    E_LevelSelector.eBoth:
        currentOrder.generatedOrder.numberOfSheets := currentOrder.order1.sheetQuantity
                                                   + currentOrder.order2.sheetQuantity;

ELSE
    // Defensive fallback (treat as Upper only)
    currentOrder.generatedOrder.numberOfSheets := currentOrder.order1.sheetQuantity;

END_CASE
END_ACTION

ACTION ACT_GenerateOrderPositions:
(*==============================================================================================================================
CPNTeck - Automação industrial
(c)Copyright 2022 All Rights Reserved
_______________________________________________________________________________________________________________________________
Library: N/A
Tested with: CX5140
Engineering: Twincat 2
Restrictions: -
Requirements: N/A
Functionality: This function block is used to generate the order positions base on the operator inputs
Support: fabio@cpnteck.com.br
Note: Parameter comments are only available in language 'English (United States)'
_______________________________________________________________________________________________________________________________
Change log table:

Version        | Date       | Expert in charge | Changes applied
01.00.01       | 29.03.2023 | Fabio Campion    | First released version
01.00.02       | 30.12.2025 | Fabio Campion    | Add E_LevelSelector selection (upper/lower/both) + fix Bottom/Top references
===============================================================================================================================*)

IF execute AND NOT executeOld THEN

    //-------------------------------------------------------------------------------------------------
    // Level selection (E_LevelSelector)
    //-------------------------------------------------------------------------------------------------
    userOrder1    := FALSE;
    useOrder2 := FALSE;

    CASE currentOrder.levelSelector OF
        E_LevelSelector.eUpperOnly:
            userOrder1    := TRUE;
            useOrder2 := FALSE;

        E_LevelSelector.eLowerOnly:
            userOrder1    := TRUE;
            useOrder2 := FALSE;

        E_LevelSelector.eBoth:
            userOrder1    := TRUE;
            useOrder2 := TRUE;

    ELSE
        // Defensive fallback
        userOrder1    := TRUE;
        useOrder2 := FALSE;
    END_CASE


    //-------------------------------------------------------------------------------------------------
    // Recalculate sheets based on selector (your method already updated previously)
    //-------------------------------------------------------------------------------------------------
    ACT_CalculateNumberOfSheets();


    (*Calculate array size*)
    toolPositionArrSize  := 30;
    knifePositionArrSize := 10;
    scorerPositionArrSize := 20;

    (*Reset positions index*)
    toolPositionIndex := 0;
    topOrderIndex     := 0;
    bottomOrderIndex  := 0;

    (*Reset positions array*)
    FOR toolPositionIndex := 1 TO toolPositionArrSize BY 1 DO
        toolPositionArr[toolPositionIndex] := 0;
    END_FOR;

    (*Reset knife positions array*)
    toolPositionIndex := 1;


    //-------------------------------------------------------------------------------------------------
    // Order totals (per level selection)
    //-------------------------------------------------------------------------------------------------
    firstOrderTotal  := 0;
    secondOrderTotal := 0;

    // TOP (Upper)
    IF userOrder1 THEN
        (*Number of boxes of the first (top) order*)
        firstOrderTotal := currentOrder.order1.sheetM1;

        (*Top order: two scorers*)
        IF (currentOrder.order1.sheetType = SHEET_WITH_TWO_SCORER)
           OR (currentOrder.order1.sheetType = SHEET_WITH_FOUR_SCORER) THEN

            firstOrderTotal := firstOrderTotal + currentOrder.order1.sheetM2;
            firstOrderTotal := firstOrderTotal + currentOrder.order1.sheetM3;
        END_IF

        (*Top order: four scorers*)
        IF currentOrder.order1.sheetType = SHEET_WITH_FOUR_SCORER THEN
            firstOrderTotal := firstOrderTotal + currentOrder.order1.sheetM4;
            firstOrderTotal := firstOrderTotal + currentOrder.order1.sheetM5;
        END_IF
    END_IF

    // BOTTOM (Lower)
    IF useOrder2 THEN
        secondOrderTotal := currentOrder.order2.sheetM1;

        (*Bottom order: two scorers*)
        IF (currentOrder.order2.sheetType = SHEET_WITH_TWO_SCORER)
           OR (currentOrder.order2.sheetType = SHEET_WITH_FOUR_SCORER) THEN

            // NOTE: corrected to Bottom (was Top in original snippet)
            secondOrderTotal := secondOrderTotal + currentOrder.order2.sheetM2;
            secondOrderTotal := secondOrderTotal + currentOrder.order2.sheetM3;
        END_IF

        (*Bottom order: four scorers*)
        IF currentOrder.order2.sheetType = SHEET_WITH_FOUR_SCORER THEN
            // NOTE: corrected to Bottom (was Top in original snippet)
            secondOrderTotal := secondOrderTotal + currentOrder.order2.sheetM4;
            secondOrderTotal := secondOrderTotal + currentOrder.order2.sheetM5;
        END_IF
    END_IF


    //-------------------------------------------------------------------------------------------------
    // Width calculations (per level selection)
    //-------------------------------------------------------------------------------------------------
    IF userOrder1 THEN
        currentOrder.generatedOrder.order1Width :=
            ( currentOrder.order1.sheetM1
            + currentOrder.order1.sheetM2
            + currentOrder.order1.sheetM3
            + currentOrder.order1.sheetM4
            + currentOrder.order1.sheetM5 ) * currentOrder.order1.sheetQuantity;
    ELSE
        currentOrder.generatedOrder.order1Width := 0;
    END_IF

    IF useOrder2 THEN
        currentOrder.generatedOrder.order2Width :=
            ( currentOrder.order2.sheetM1
            + currentOrder.order2.sheetM2
            + currentOrder.order2.sheetM3
            + currentOrder.order2.sheetM4
            + currentOrder.order2.sheetM5 ) * currentOrder.order2.sheetQuantity;
    ELSE
        currentOrder.generatedOrder.order2Width := 0;
    END_IF

    currentOrder.generatedOrder.orderTotalWidth :=
        currentOrder.generatedOrder.order1Width + currentOrder.generatedOrder.order2Width;

    firstKnifePosition := (machineConfig.machineWidth - currentOrder.generatedOrder.orderTotalWidth) / 2;


    //-------------------------------------------------------------------------------------------------
    // Tool position generation
    //-------------------------------------------------------------------------------------------------
    (*First Knife position*)
    toolPositionArr[toolPositionIndex] := firstKnifePosition; // The first knife always uses the first position
    toolPositionIndex := toolPositionIndex + 1;

    // TOP order positions
    IF userOrder1 THEN
        FOR topOrderIndex := 1 TO currentOrder.order1.sheetQuantity BY 1 DO

            (*Box without scorer*)
            toolPositionArr[toolPositionIndex] := firstKnifePosition + currentOrder.order1.sheetM1;
            firstKnifePosition := firstKnifePosition + currentOrder.order1.sheetM1;
            toolPositionIndex := toolPositionIndex + 1;

            (*Box with two scorers*)
            IF (currentOrder.order1.sheetType = SHEET_WITH_TWO_SCORER)
               OR (currentOrder.order1.sheetType = SHEET_WITH_FOUR_SCORER) THEN

                toolPositionArr[toolPositionIndex] := firstKnifePosition + currentOrder.order1.sheetM2;
                firstKnifePosition := firstKnifePosition + currentOrder.order1.sheetM2;
                toolPositionIndex := toolPositionIndex + 1;

                toolPositionArr[toolPositionIndex] := firstKnifePosition + currentOrder.order1.sheetM3;
                firstKnifePosition := firstKnifePosition + currentOrder.order1.sheetM3;
                toolPositionIndex := toolPositionIndex + 1;
            END_IF

            (*Box with 4 scorers*)
            IF currentOrder.order1.sheetType = SHEET_WITH_FOUR_SCORER THEN

                toolPositionArr[toolPositionIndex] := firstKnifePosition + currentOrder.order1.sheetM4;
                firstKnifePosition := firstKnifePosition + currentOrder.order1.sheetM4;
                toolPositionIndex := toolPositionIndex + 1;

                toolPositionArr[toolPositionIndex] := firstKnifePosition + currentOrder.order1.sheetM5;
                firstKnifePosition := firstKnifePosition + currentOrder.order1.sheetM5;
                toolPositionIndex := toolPositionIndex + 1;
            END_IF

        END_FOR
    END_IF

    // BOTTOM order positions
    IF useOrder2 THEN
        FOR bottomOrderIndex := 1 TO currentOrder.order2.sheetQuantity BY 1 DO

            (*Box without scorer*)
            toolPositionArr[toolPositionIndex] := firstKnifePosition + currentOrder.order2.sheetM1;
            firstKnifePosition := firstKnifePosition + currentOrder.order2.sheetM1;
            toolPositionIndex := toolPositionIndex + 1;

            (*Box with two scorers*)
            IF (currentOrder.order2.sheetType = SHEET_WITH_TWO_SCORER)
               OR (currentOrder.order2.sheetType = SHEET_WITH_FOUR_SCORER) THEN

                toolPositionArr[toolPositionIndex] := firstKnifePosition + currentOrder.order2.sheetM2;
                firstKnifePosition := firstKnifePosition + currentOrder.order2.sheetM2;
                toolPositionIndex := toolPositionIndex + 1;

                toolPositionArr[toolPositionIndex] := firstKnifePosition + currentOrder.order2.sheetM3;
                firstKnifePosition := firstKnifePosition + currentOrder.order2.sheetM3;
                toolPositionIndex := toolPositionIndex + 1;
            END_IF

            (*Box with 4 scorers*)
            IF currentOrder.order2.sheetType = SHEET_WITH_FOUR_SCORER THEN

                toolPositionArr[toolPositionIndex] := firstKnifePosition + currentOrder.order2.sheetM4;
                firstKnifePosition := firstKnifePosition + currentOrder.order2.sheetM4;
                toolPositionIndex := toolPositionIndex + 1;

                toolPositionArr[toolPositionIndex] := firstKnifePosition + currentOrder.order2.sheetM5;
                firstKnifePosition := firstKnifePosition + currentOrder.order2.sheetM5;
                toolPositionIndex := toolPositionIndex + 1;
            END_IF

        END_FOR
    END_IF


    //-------------------------------------------------------------------------------------------------
    // Post-processing (unchanged call flow)
    //-------------------------------------------------------------------------------------------------
    ACT_CalculateNumberOfKnifes();
    ACT_KnifePositionSelection();  // Call the program
    ACT_ScorerPositionSelection(); // Call the program

END_IF

executeOld := execute;
END_ACTION

ACTION ACT_KnifePositionDistribution:
(*==============================================================================================================================
CPNTeck - Automação industrial - MRBrasil Refactored
Version: 01.00.04 | Date: 19.02.2026 | Expert: Gemini AI
Functionality: Optimized position distribution with DYNAMIC boundary detection.
===============================================================================================================================

// 1. Reset all Enables to FALSE and clear boundaries
FOR i := 1 TO 5 DO
	currentOrder.generatedOrder.knifeEnabledArr[i] := FALSE;
END_FOR

currentOrder.generatedOrder.firstKnifePosition := 0.0;
currentOrder.generatedOrder.lastKnifePosition  := 0.0;

// 2. Position Distribution (MRBrasil specific logic)
CASE currentOrder.generatedOrder.numberOfKnifes OF

	2:
		currentOrder.generatedOrder.knifeEnabledArr[1] := TRUE;
		currentOrder.generatedOrder.knifeEnabledArr[5] := TRUE;
		
		currentOrder.generatedOrder.knifePositionReferenceArr[1] := knifePositionArr[1];
		currentOrder.generatedOrder.knifePositionReferenceArr[2] := knifePositionArr[1] + 150;
		currentOrder.generatedOrder.knifePositionReferenceArr[3] := knifePositionArr[1] + 300;
		currentOrder.generatedOrder.knifePositionReferenceArr[4] := knifePositionArr[2] - 150;
		currentOrder.generatedOrder.knifePositionReferenceArr[5] := knifePositionArr[2];

	3:
		IF knifePositionArr[2] > machineConfig.knifeMaxPostionArr[3] THEN
			currentOrder.generatedOrder.knifeEnabledArr[1] := TRUE;
			currentOrder.generatedOrder.knifeEnabledArr[4] := TRUE;
			currentOrder.generatedOrder.knifeEnabledArr[5] := TRUE;
			
			currentOrder.generatedOrder.knifePositionReferenceArr[1] := knifePositionArr[1];
			currentOrder.generatedOrder.knifePositionReferenceArr[2] := knifePositionArr[1] + 150;
			currentOrder.generatedOrder.knifePositionReferenceArr[3] := knifePositionArr[1] + 300;
			currentOrder.generatedOrder.knifePositionReferenceArr[4] := knifePositionArr[2];
			currentOrder.generatedOrder.knifePositionReferenceArr[5] := knifePositionArr[3];
		ELSE
			currentOrder.generatedOrder.knifeEnabledArr[1] := TRUE;
			currentOrder.generatedOrder.knifeEnabledArr[3] := TRUE;
			currentOrder.generatedOrder.knifeEnabledArr[5] := TRUE;
			
			currentOrder.generatedOrder.knifePositionReferenceArr[1] := knifePositionArr[1];
			currentOrder.generatedOrder.knifePositionReferenceArr[2] := knifePositionArr[1] + 150;
			currentOrder.generatedOrder.knifePositionReferenceArr[3] := knifePositionArr[2];
			currentOrder.generatedOrder.knifePositionReferenceArr[4] := knifePositionArr[3] - 150;
			currentOrder.generatedOrder.knifePositionReferenceArr[5] := knifePositionArr[3];
		END_IF

	4:
		IF knifePositionArr[3] > machineConfig.knifeMaxPostionArr[3] THEN
			currentOrder.generatedOrder.knifeEnabledArr[1] := TRUE;
			currentOrder.generatedOrder.knifeEnabledArr[2] := TRUE;
			currentOrder.generatedOrder.knifeEnabledArr[4] := TRUE;
			currentOrder.generatedOrder.knifeEnabledArr[5] := TRUE;
			
			currentOrder.generatedOrder.knifePositionReferenceArr[1] := knifePositionArr[1];
			currentOrder.generatedOrder.knifePositionReferenceArr[2] := knifePositionArr[2];
			currentOrder.generatedOrder.knifePositionReferenceArr[3] := knifePositionArr[2] + 150;
			currentOrder.generatedOrder.knifePositionReferenceArr[4] := knifePositionArr[3];
			currentOrder.generatedOrder.knifePositionReferenceArr[5] := knifePositionArr[4];
		ELSE
			currentOrder.generatedOrder.knifeEnabledArr[1] := TRUE;
			currentOrder.generatedOrder.knifeEnabledArr[2] := TRUE;
			currentOrder.generatedOrder.knifeEnabledArr[3] := TRUE;
			currentOrder.generatedOrder.knifeEnabledArr[5] := TRUE;
			
			currentOrder.generatedOrder.knifePositionReferenceArr[1] := knifePositionArr[1];
			currentOrder.generatedOrder.knifePositionReferenceArr[2] := knifePositionArr[2];
			currentOrder.generatedOrder.knifePositionReferenceArr[3] := knifePositionArr[3];
			currentOrder.generatedOrder.knifePositionReferenceArr[4] := knifePositionArr[4] - 150;
			currentOrder.generatedOrder.knifePositionReferenceArr[5] := knifePositionArr[4];
		END_IF

	5:
		FOR i := 1 TO 5 DO
			currentOrder.generatedOrder.knifeEnabledArr[i] := TRUE;
			currentOrder.generatedOrder.knifePositionReferenceArr[i] := knifePositionArr[i];
		END_FOR

END_CASE

// 3. DYNAMIC BOUNDARY DETECTION
// Find the first enabled knife
FOR i := 1 TO 5 DO
    IF currentOrder.generatedOrder.knifeEnabledArr[i] THEN
        currentOrder.generatedOrder.firstKnifePosition := currentOrder.generatedOrder.knifePositionReferenceArr[i];
        EXIT; // Stop at the first one found
    END_IF
END_FOR

// Find the last enabled knife
FOR i := 5 TO 1 BY -1 DO
    IF currentOrder.generatedOrder.knifeEnabledArr[i] THEN
        currentOrder.generatedOrder.lastKnifePosition := currentOrder.generatedOrder.knifePositionReferenceArr[i];
        EXIT; // Stop at the last one found (searching backwards)
    END_IF
END_FOR
*)


(*==============================================================================================================================
CPNTeck - Automação industrial
(c)Copyright 2022 All Rights Reserved
_______________________________________________________________________________________________________________________________
Library: N/A 
Tested with: CX5140
Engineering: Twincat 2
Restrictions: -
Requirements: N/A
Functionality: This function block is used to distribute the position for the desired knife
Support: fabio@cpnteck.com.br
Note: Parameter comments are only available in language 'English (United States)'
_______________________________________________________________________________________________________________________________
Change log table:

Version  		| Date        			| Expert in charge  	| Changes applied
01.00.01		| 29.03.2023  		| Fabio Campion            | First released version



===============================================================================================================================*)

IF currentOrder.generatedOrder.numberOfKnifes = 2 THEN

	currentOrder.generatedOrder.knifeEnabledArr[01] := TRUE;
	currentOrder.generatedOrder.knifeEnabledArr[02] := FALSE;
	currentOrder.generatedOrder.knifeEnabledArr[03] := FALSE;
	currentOrder.generatedOrder.knifeEnabledArr[04] := FALSE;
	currentOrder.generatedOrder.knifeEnabledArr[05] := TRUE;

	currentOrder.generatedOrder.knifePositionReferenceArr[1] := knifePositionArr[1];
	currentOrder.generatedOrder.knifePositionReferenceArr[2] := knifePositionArr[1] + 160;
	currentOrder.generatedOrder.knifePositionReferenceArr[3] := knifePositionArr[1] + 160 + 160;
	currentOrder.generatedOrder.knifePositionReferenceArr[4] := knifePositionArr[2] - 160;
	currentOrder.generatedOrder.knifePositionReferenceArr[5] := knifePositionArr[2];

END_IF

IF currentOrder.generatedOrder.numberOfKnifes = 3 THEN


	IF knifePositionArr[2] > machineConfig.knifeMaxPostionArr[3] THEN
		
		currentOrder.generatedOrder.knifeEnabledArr[01] := TRUE;
		currentOrder.generatedOrder.knifeEnabledArr[02] := FALSE;
		currentOrder.generatedOrder.knifeEnabledArr[03] := FALSE;
		currentOrder.generatedOrder.knifeEnabledArr[04] := TRUE;
		currentOrder.generatedOrder.knifeEnabledArr[05] := TRUE;
	
		currentOrder.generatedOrder.knifePositionReferenceArr[1] := knifePositionArr[1];
		currentOrder.generatedOrder.knifePositionReferenceArr[2] := knifePositionArr[1] + 160;
		currentOrder.generatedOrder.knifePositionReferenceArr[3] := knifePositionArr[1] + 160 + 160;
		currentOrder.generatedOrder.knifePositionReferenceArr[4] := knifePositionArr[2];
		currentOrder.generatedOrder.knifePositionReferenceArr[5] := knifePositionArr[3];
	
	ELSE
		
		currentOrder.generatedOrder.knifeEnabledArr[01] := TRUE;
		currentOrder.generatedOrder.knifeEnabledArr[02] := FALSE;
		currentOrder.generatedOrder.knifeEnabledArr[03] := TRUE;
		currentOrder.generatedOrder.knifeEnabledArr[04] := FALSE;
		currentOrder.generatedOrder.knifeEnabledArr[05] := TRUE;
	
		currentOrder.generatedOrder.knifePositionReferenceArr[1] := knifePositionArr[1];
		currentOrder.generatedOrder.knifePositionReferenceArr[2] := knifePositionArr[1] + 160;
		currentOrder.generatedOrder.knifePositionReferenceArr[3] := knifePositionArr[2];
		currentOrder.generatedOrder.knifePositionReferenceArr[4] := knifePositionArr[3] - 160;
		currentOrder.generatedOrder.knifePositionReferenceArr[5] := knifePositionArr[3];
		
	END_IF
END_IF

IF currentOrder.generatedOrder.numberOfKnifes = 4 THEN

	IF knifePositionArr[3] > machineConfig.knifeMaxPostionArr[3] THEN
		
		currentOrder.generatedOrder.knifeEnabledArr[01] := TRUE;
		currentOrder.generatedOrder.knifeEnabledArr[02] := TRUE;
		currentOrder.generatedOrder.knifeEnabledArr[03] := FALSE;
		currentOrder.generatedOrder.knifeEnabledArr[04] := TRUE;
		currentOrder.generatedOrder.knifeEnabledArr[05] := TRUE;
	
		currentOrder.generatedOrder.knifePositionReferenceArr[1] := knifePositionArr[1];
		currentOrder.generatedOrder.knifePositionReferenceArr[2] := knifePositionArr[2];
		currentOrder.generatedOrder.knifePositionReferenceArr[3] := knifePositionArr[2] + 160;
		currentOrder.generatedOrder.knifePositionReferenceArr[4] := knifePositionArr[3];
		currentOrder.generatedOrder.knifePositionReferenceArr[5] := knifePositionArr[4];		
		
	ELSE
		
		currentOrder.generatedOrder.knifeEnabledArr[01] := TRUE;
		currentOrder.generatedOrder.knifeEnabledArr[02] := TRUE;
		currentOrder.generatedOrder.knifeEnabledArr[03] := TRUE;
		currentOrder.generatedOrder.knifeEnabledArr[04] := FALSE;
		currentOrder.generatedOrder.knifeEnabledArr[05] := TRUE;
	
		currentOrder.generatedOrder.knifePositionReferenceArr[1] := knifePositionArr[1];
		currentOrder.generatedOrder.knifePositionReferenceArr[2] := knifePositionArr[2];
		currentOrder.generatedOrder.knifePositionReferenceArr[3] := knifePositionArr[3];
		currentOrder.generatedOrder.knifePositionReferenceArr[4] := knifePositionArr[4] - 160;
		currentOrder.generatedOrder.knifePositionReferenceArr[5] := knifePositionArr[4];		
		
	END_IF

	
	
	
	
END_IF

IF currentOrder.generatedOrder.numberOfKnifes = 5 THEN

	currentOrder.generatedOrder.knifeEnabledArr[01] := TRUE;
	currentOrder.generatedOrder.knifeEnabledArr[02] := TRUE;
	currentOrder.generatedOrder.knifeEnabledArr[03] := TRUE;
	currentOrder.generatedOrder.knifeEnabledArr[04] := TRUE;
	currentOrder.generatedOrder.knifeEnabledArr[05] := TRUE;

	currentOrder.generatedOrder.knifePositionReferenceArr[1] := knifePositionArr[1];
	currentOrder.generatedOrder.knifePositionReferenceArr[2] := knifePositionArr[2];
	currentOrder.generatedOrder.knifePositionReferenceArr[3] := knifePositionArr[3];
	currentOrder.generatedOrder.knifePositionReferenceArr[4] := knifePositionArr[4];
	currentOrder.generatedOrder.knifePositionReferenceArr[5] := knifePositionArr[5];

END_IF
END_ACTION

ACTION ACT_KnifePositionDistribution_bak:

(*==============================================================================================================================
CPNTeck - Automação industrial
(c)Copyright 2022 All Rights Reserved
_______________________________________________________________________________________________________________________________
Library: N/A 
Tested with: CX5140
Engineering: Twincat 2
Restrictions: -
Requirements: N/A
Functionality: This function block is used to distribute the position for the desired knife
Support: fabio@cpnteck.com.br
Note: Parameter comments are only available in language 'English (United States)'
_______________________________________________________________________________________________________________________________
Change log table:

Version  		| Date        			| Expert in charge  	| Changes applied
01.00.01		| 29.03.2023  		| Fabio Campion            | First released version



===============================================================================================================================*)

IF currentOrder.generatedOrder.numberOfKnifes = 2 THEN

	currentOrder.generatedOrder.knifeEnabledArr[01] := TRUE;
	currentOrder.generatedOrder.knifeEnabledArr[02] := FALSE;
	currentOrder.generatedOrder.knifeEnabledArr[03] := FALSE;
	currentOrder.generatedOrder.knifeEnabledArr[04] := FALSE;
	currentOrder.generatedOrder.knifeEnabledArr[05] := TRUE;

	currentOrder.generatedOrder.knifePositionReferenceArr[1] := knifePositionArr[1];
	currentOrder.generatedOrder.knifePositionReferenceArr[2] := knifePositionArr[1] + 150;
	currentOrder.generatedOrder.knifePositionReferenceArr[3] := knifePositionArr[1] + 150 + 150;
	currentOrder.generatedOrder.knifePositionReferenceArr[4] := knifePositionArr[2] - 150;
	currentOrder.generatedOrder.knifePositionReferenceArr[5] := knifePositionArr[2];

END_IF

IF currentOrder.generatedOrder.numberOfKnifes = 3 THEN


	IF knifePositionArr[2] > machineConfig.knifeMaxPostionArr[3] THEN
		
		currentOrder.generatedOrder.knifeEnabledArr[01] := TRUE;
		currentOrder.generatedOrder.knifeEnabledArr[02] := FALSE;
		currentOrder.generatedOrder.knifeEnabledArr[03] := FALSE;
		currentOrder.generatedOrder.knifeEnabledArr[04] := TRUE;
		currentOrder.generatedOrder.knifeEnabledArr[05] := TRUE;
	
		currentOrder.generatedOrder.knifePositionReferenceArr[1] := knifePositionArr[1];
		currentOrder.generatedOrder.knifePositionReferenceArr[2] := knifePositionArr[1] + 150;
		currentOrder.generatedOrder.knifePositionReferenceArr[3] := knifePositionArr[1] + 150 + 150;
		currentOrder.generatedOrder.knifePositionReferenceArr[4] := knifePositionArr[2];
		currentOrder.generatedOrder.knifePositionReferenceArr[5] := knifePositionArr[3];
	
	ELSE
		
		currentOrder.generatedOrder.knifeEnabledArr[01] := TRUE;
		currentOrder.generatedOrder.knifeEnabledArr[02] := FALSE;
		currentOrder.generatedOrder.knifeEnabledArr[03] := TRUE;
		currentOrder.generatedOrder.knifeEnabledArr[04] := FALSE;
		currentOrder.generatedOrder.knifeEnabledArr[05] := TRUE;
	
		currentOrder.generatedOrder.knifePositionReferenceArr[1] := knifePositionArr[1];
		currentOrder.generatedOrder.knifePositionReferenceArr[2] := knifePositionArr[1] + 150;
		currentOrder.generatedOrder.knifePositionReferenceArr[3] := knifePositionArr[2];
		currentOrder.generatedOrder.knifePositionReferenceArr[4] := knifePositionArr[3] - 150;
		currentOrder.generatedOrder.knifePositionReferenceArr[5] := knifePositionArr[3];
		
	END_IF
END_IF

IF currentOrder.generatedOrder.numberOfKnifes = 4 THEN

	IF knifePositionArr[3] > machineConfig.knifeMaxPostionArr[3] THEN
		
		currentOrder.generatedOrder.knifeEnabledArr[01] := TRUE;
		currentOrder.generatedOrder.knifeEnabledArr[02] := TRUE;
		currentOrder.generatedOrder.knifeEnabledArr[03] := FALSE;
		currentOrder.generatedOrder.knifeEnabledArr[04] := TRUE;
		currentOrder.generatedOrder.knifeEnabledArr[05] := TRUE;
	
		currentOrder.generatedOrder.knifePositionReferenceArr[1] := knifePositionArr[1];
		currentOrder.generatedOrder.knifePositionReferenceArr[2] := knifePositionArr[2];
		currentOrder.generatedOrder.knifePositionReferenceArr[3] := knifePositionArr[2] + 150;
		currentOrder.generatedOrder.knifePositionReferenceArr[4] := knifePositionArr[3];
		currentOrder.generatedOrder.knifePositionReferenceArr[5] := knifePositionArr[4];		
		
	ELSE
		
		currentOrder.generatedOrder.knifeEnabledArr[01] := TRUE;
		currentOrder.generatedOrder.knifeEnabledArr[02] := TRUE;
		currentOrder.generatedOrder.knifeEnabledArr[03] := TRUE;
		currentOrder.generatedOrder.knifeEnabledArr[04] := FALSE;
		currentOrder.generatedOrder.knifeEnabledArr[05] := TRUE;
	
		currentOrder.generatedOrder.knifePositionReferenceArr[1] := knifePositionArr[1];
		currentOrder.generatedOrder.knifePositionReferenceArr[2] := knifePositionArr[2];
		currentOrder.generatedOrder.knifePositionReferenceArr[3] := knifePositionArr[3];
		currentOrder.generatedOrder.knifePositionReferenceArr[4] := knifePositionArr[4] - 150;
		currentOrder.generatedOrder.knifePositionReferenceArr[5] := knifePositionArr[4];		
		
	END_IF

	
	
	
	
END_IF

IF currentOrder.generatedOrder.numberOfKnifes = 5 THEN

	currentOrder.generatedOrder.knifeEnabledArr[01] := TRUE;
	currentOrder.generatedOrder.knifeEnabledArr[02] := TRUE;
	currentOrder.generatedOrder.knifeEnabledArr[03] := TRUE;
	currentOrder.generatedOrder.knifeEnabledArr[04] := TRUE;
	currentOrder.generatedOrder.knifeEnabledArr[05] := TRUE;

	currentOrder.generatedOrder.knifePositionReferenceArr[1] := knifePositionArr[1];
	currentOrder.generatedOrder.knifePositionReferenceArr[2] := knifePositionArr[2];
	currentOrder.generatedOrder.knifePositionReferenceArr[3] := knifePositionArr[3];
	currentOrder.generatedOrder.knifePositionReferenceArr[4] := knifePositionArr[4];
	currentOrder.generatedOrder.knifePositionReferenceArr[5] := knifePositionArr[5];

END_IF
END_ACTION

ACTION ACT_KnifePositionSelection:
(*==============================================================================================================================
CPNTeck - Automação industrial
(c)Copyright 2022 All Rights Reserved
_______________________________________________________________________________________________________________________________
Library: N/A
Tested with: CX5140
Engineering: Twincat 2
Restrictions: -
Requirements: N/A
Functionality:
    Distribute knife positions from toolPositionArr[] into knifePositionArr[] according to:
      - Sheet type (0 / 2 / 4 scorers) => step size (1 / 3 / 5)
      - E_LevelSelector => UpperOnly / LowerOnly / Both
Support: fabio@cpnteck.com.br
Note: Parameter comments are only available in language 'English (United States)'
_______________________________________________________________________________________________________________________________
Change log table:
Version        | Date       | Expert in charge | Changes applied
01.00.01       | 29.03.2023 | Fabio Campion    | First released version
01.00.02       | 30.12.2025 | Fabio Campion    | Add E_LevelSelector selection (upper/lower/both) + fix index handling
===============================================================================================================================*)
{region "Knife Position Selection — Reset arrays"}

(* Reset the knife enabled/position arrays (knives are 1..7 in your project) *)
FOR knifeEnabledIndex := 1 TO 7 BY 1 DO
    currentOrder.generatedOrder.knifeEnabledArr[knifeEnabledIndex] := FALSE;
    knifePositionArr[knifeEnabledIndex] := 0;
    currentOrder.generatedOrder.knifePositionReferenceArr[knifeEnabledIndex] := 0;
END_FOR;

(* Reset distribution indexes *)
knifeDistributionIndex := 1;  // Index into toolPositionArr[]
knifeOutIdx            := 1;  // Index into knifePositionArr[]

{endregion}


{region "Knife Position Selection — Determine active levels (E_LevelSelector)"}

userOrder1    := FALSE;
useOrder2 := FALSE;

CASE currentOrder.levelSelector OF
    E_LevelSelector.eUpperOnly:
        userOrder1    := TRUE;
        useOrder2 := FALSE;

    E_LevelSelector.eLowerOnly:
        userOrder1    := TRUE;
        useOrder2 := FALSE;

    E_LevelSelector.eBoth:
        userOrder1    := TRUE;
        useOrder2 := TRUE;

ELSE
    // Defensive fallback: keep legacy behavior (Top only)
    userOrder1    := TRUE;
    useOrder2 := FALSE;
END_CASE

{endregion}


{region "Knife Position Selection — TOP distribution"}

IF userOrder1 THEN

    topStep := 1;
    CASE currentOrder.order1.sheetType OF
        SHEET_WITH_NO_SCORER:   topStep := 1;
        SHEET_WITH_TWO_SCORER:  topStep := 3;
        SHEET_WITH_FOUR_SCORER: topStep := 5;
    ELSE
        topStep := 1;
    END_CASE

    // For each produced sheet, take one knife position then jump by step
    FOR knifePositionTopIndex := 1 TO currentOrder.order1.sheetQuantity BY 1 DO
        knifePositionArr[knifeOutIdx] := toolPositionArr[knifeDistributionIndex];
        knifeOutIdx := knifeOutIdx + 1;
        knifeDistributionIndex := knifeDistributionIndex + topStep;
    END_FOR

    // Final knife after last top box (end of top order)
    knifePositionArr[knifeOutIdx] := toolPositionArr[knifeDistributionIndex];
    knifeOutIdx := knifeOutIdx + 1;

END_IF

{endregion}


{region "Knife Position Selection — BOTTOM distribution"}

IF useOrder2 THEN

    bottomStep := 1;
    CASE currentOrder.order2.sheetType OF
        SHEET_WITH_NO_SCORER:   bottomStep := 1;
        SHEET_WITH_TWO_SCORER:  bottomStep := 3;
        SHEET_WITH_FOUR_SCORER: bottomStep := 5;
    ELSE
        bottomStep := 1;
    END_CASE

    // If TOP and BOTTOM are enabled, the start knife of bottom equals the last knife of top.
    // Therefore, DO NOT write the shared boundary again.
    IF userOrder1 THEN

        // BOTH enabled: write only END-OF-SHEET knives for bottom
        FOR knifePositionBottomIndex := 1 TO currentOrder.order2.sheetQuantity BY 1 DO
            knifeDistributionIndex := knifeDistributionIndex + bottomStep;          // move to end-of-sheet
            knifePositionArr[knifeOutIdx] := toolPositionArr[knifeDistributionIndex];
            knifeOutIdx := knifeOutIdx + 1;
        END_FOR

    ELSE

        // BOTTOM only: legacy behavior (start + final)
        FOR knifePositionBottomIndex := 1 TO currentOrder.order2.sheetQuantity BY 1 DO
            knifePositionArr[knifeOutIdx] := toolPositionArr[knifeDistributionIndex];
            knifeOutIdx := knifeOutIdx + 1;
            knifeDistributionIndex := knifeDistributionIndex + bottomStep;
        END_FOR

        // Final knife after last bottom box
        knifePositionArr[knifeOutIdx] := toolPositionArr[knifeDistributionIndex];
        knifeOutIdx := knifeOutIdx + 1;

    END_IF

END_IF

ACT_KnifePositionDistribution();
	 
{endregion}
END_ACTION

ACTION ACT_ScorerPositionDistribution:
(*===============================================================================================================================
CPNTeck - Automação Industrial
(c)Copyright 2022-2025 All Rights Reserved
_______________________________________________________________________________________________________________________________
Functionality: Scorer Distribution Logic (Merged Version)
Target: MRBRASIL Logic with COCELPA Variable Naming
_______________________________________________________________________________________________________________________________
Change log table:
Version      | Date          | Expert in charge | Changes applied
01.00.05     | 17.02.2026   | Gemini AI        | Merged MRBRASIL logic into COCELPA naming structure
                                               | (Uses .order1/.order2 and active Home positioning)
===============================================================================================================================*)

// Verifica se ambos os pedidos não possuem vincadores
IF currentOrder.order1.sheetType = SHEET_WITH_NO_SCORER AND currentOrder.order2.sheetType = SHEET_WITH_NO_SCORER THEN
    // Lógica MRBRASIL: Envia para home E desabilita
    FOR i := 1 TO 8 DO
        currentOrder.generatedOrder.scorerPositionReferenceArr[i] := machineConfig.homePositionScorer[i];
        currentOrder.generatedOrder.scorerEnabledArr[i] := FALSE;
    END_FOR

ELSE
    // Default: Reset preventivo para Home (Comportamento MRBRASIL)
    FOR i := 1 TO 8 DO
        currentOrder.generatedOrder.scorerPositionReferenceArr[i] := machineConfig.homePositionScorer[i];
        currentOrder.generatedOrder.scorerEnabledArr[i] := FALSE;
    END_FOR

    //──────────────────────────────────────────────────────────────────────────────
    // Top Order Logic (Usando .order1 da COCELPA)
    //──────────────────────────────────────────────────────────────────────────────
    CASE currentOrder.order1.sheetQuantity OF
        1:
            CASE currentOrder.order1.sheetType OF
                SHEET_WITH_TWO_SCORER:
                    // Option 1: Scorer 3 e 4
                    IF NOT (scorerPositionArr[1] > machineConfig.scorerMaxPostionArr[3] OR
                        scorerPositionArr[2] > machineConfig.scorerMaxPostionArr[4] OR
                        scorerPositionArr[1] < machineConfig.scorerMinPostionArr[3] OR
                        scorerPositionArr[2] < machineConfig.scorerMinPostionArr[4]) THEN
                        currentOrder.generatedOrder.scorerPositionReferenceArr[3] := scorerPositionArr[1];
                        currentOrder.generatedOrder.scorerPositionReferenceArr[4] := scorerPositionArr[2];
                        currentOrder.generatedOrder.scorerEnabledArr[3] := TRUE;
                        currentOrder.generatedOrder.scorerEnabledArr[4] := TRUE;
                
                    // Option 2: Scorer 5 e 6
                    ELSIF NOT (scorerPositionArr[1] > machineConfig.scorerMaxPostionArr[5] OR
                        scorerPositionArr[2] > machineConfig.scorerMaxPostionArr[6] OR
                        scorerPositionArr[1] < machineConfig.scorerMinPostionArr[5] OR
                        scorerPositionArr[2] < machineConfig.scorerMinPostionArr[6]) THEN
                        currentOrder.generatedOrder.scorerPositionReferenceArr[5] := scorerPositionArr[1];
                        currentOrder.generatedOrder.scorerPositionReferenceArr[6] := scorerPositionArr[2];
                        currentOrder.generatedOrder.scorerEnabledArr[5] := TRUE;
                        currentOrder.generatedOrder.scorerEnabledArr[6] := TRUE;
                
                    // Option 3: Scorer 3 e 5
                    ELSIF NOT (scorerPositionArr[1] > machineConfig.scorerMaxPostionArr[3] OR
                        scorerPositionArr[2] > machineConfig.scorerMaxPostionArr[5] OR
                        scorerPositionArr[1] < machineConfig.scorerMinPostionArr[3] OR
                        scorerPositionArr[2] < machineConfig.scorerMinPostionArr[5]) THEN
                        currentOrder.generatedOrder.scorerPositionReferenceArr[3] := scorerPositionArr[1];
                        currentOrder.generatedOrder.scorerPositionReferenceArr[5] := scorerPositionArr[2];
                        currentOrder.generatedOrder.scorerEnabledArr[3] := TRUE;
                        currentOrder.generatedOrder.scorerEnabledArr[5] := TRUE;
                
                    // Option 4: Scorer 4 e 6
                    ELSIF NOT (scorerPositionArr[1] > machineConfig.scorerMaxPostionArr[4] OR
                        scorerPositionArr[2] > machineConfig.scorerMaxPostionArr[6] OR
                        scorerPositionArr[1] < machineConfig.scorerMinPostionArr[4] OR
                        scorerPositionArr[2] < machineConfig.scorerMinPostionArr[6]) THEN
                        currentOrder.generatedOrder.scorerPositionReferenceArr[4] := scorerPositionArr[1];
                        currentOrder.generatedOrder.scorerPositionReferenceArr[6] := scorerPositionArr[2];
                        currentOrder.generatedOrder.scorerEnabledArr[4] := TRUE;
                        currentOrder.generatedOrder.scorerEnabledArr[6] := TRUE;
                
                    // Option 5: Scorer 1 e 2 (+ aux 150mm)
                    ELSIF NOT (scorerPositionArr[1] > machineConfig.scorerMaxPostionArr[1] OR
                        scorerPositionArr[2] > machineConfig.scorerMaxPostionArr[2] OR
                        scorerPositionArr[1] + 150 > machineConfig.scorerMaxPostionArr[3] OR
                        scorerPositionArr[2] + 150 > machineConfig.scorerMaxPostionArr[4] OR
                        scorerPositionArr[1] < machineConfig.scorerMinPostionArr[1] OR
                        scorerPositionArr[2] < machineConfig.scorerMinPostionArr[2]) THEN
                        currentOrder.generatedOrder.scorerPositionReferenceArr[1] := scorerPositionArr[1];
                        currentOrder.generatedOrder.scorerPositionReferenceArr[2] := scorerPositionArr[2];
                        currentOrder.generatedOrder.scorerPositionReferenceArr[3] := scorerPositionArr[1] + 160;
                        currentOrder.generatedOrder.scorerPositionReferenceArr[4] := scorerPositionArr[2] + 160;
                        currentOrder.generatedOrder.scorerEnabledArr[1] := TRUE;
                        currentOrder.generatedOrder.scorerEnabledArr[2] := TRUE;
                
                    // Option 6: Scorer 1 e 3
                    ELSIF NOT (scorerPositionArr[1] > machineConfig.scorerMaxPostionArr[1] OR
                        scorerPositionArr[2] > machineConfig.scorerMaxPostionArr[3] OR
                        scorerPositionArr[1] < machineConfig.scorerMinPostionArr[1] OR
                        scorerPositionArr[2] < machineConfig.scorerMinPostionArr[3]) THEN
                        currentOrder.generatedOrder.scorerPositionReferenceArr[1] := scorerPositionArr[1];
                        currentOrder.generatedOrder.scorerPositionReferenceArr[3] := scorerPositionArr[2];
                        currentOrder.generatedOrder.scorerEnabledArr[1] := TRUE;
                        currentOrder.generatedOrder.scorerEnabledArr[3] := TRUE;
                
                    // Option 7: Scorer 2 e 4
                    ELSIF NOT (scorerPositionArr[1] > machineConfig.scorerMaxPostionArr[2] OR
                        scorerPositionArr[2] > machineConfig.scorerMaxPostionArr[4] OR
                        scorerPositionArr[1] < machineConfig.scorerMinPostionArr[2] OR
                        scorerPositionArr[2] < machineConfig.scorerMinPostionArr[4]) THEN
                        currentOrder.generatedOrder.scorerPositionReferenceArr[2] := scorerPositionArr[1];
                        currentOrder.generatedOrder.scorerPositionReferenceArr[4] := scorerPositionArr[2];
                        currentOrder.generatedOrder.scorerEnabledArr[2] := TRUE;
                        currentOrder.generatedOrder.scorerEnabledArr[4] := TRUE;
                    END_IF;

                SHEET_WITH_FOUR_SCORER:
                    FOR i := 1 TO 4 DO
                        currentOrder.generatedOrder.scorerPositionReferenceArr[i] := scorerPositionArr[i];
                        currentOrder.generatedOrder.scorerEnabledArr[i] := TRUE;
                    END_FOR;
            END_CASE;

        2:
            CASE currentOrder.order1.sheetType OF
                SHEET_WITH_TWO_SCORER:
                    FOR i := 1 TO 4 DO
                        currentOrder.generatedOrder.scorerPositionReferenceArr[i] := scorerPositionArr[i];
                        currentOrder.generatedOrder.scorerEnabledArr[i] := TRUE;
                    END_FOR;
                SHEET_WITH_FOUR_SCORER:
                    FOR i := 1 TO 8 DO
                        currentOrder.generatedOrder.scorerPositionReferenceArr[i] := scorerPositionArr[i];
                        currentOrder.generatedOrder.scorerEnabledArr[i] := TRUE;
                    END_FOR;
            END_CASE;

        3:
            FOR i := 1 TO 6 DO
                currentOrder.generatedOrder.scorerPositionReferenceArr[i + 1] := scorerPositionArr[i];
                currentOrder.generatedOrder.scorerEnabledArr[i + 1] := TRUE;
            END_FOR;

        4, 5:
            FOR i := 1 TO 8 DO
                currentOrder.generatedOrder.scorerPositionReferenceArr[i] := scorerPositionArr[i];
                currentOrder.generatedOrder.scorerEnabledArr[i] := TRUE;
            END_FOR;
    END_CASE;

    //──────────────────────────────────────────────────────────────────────────────
    // Bottom Order Logic (Usando .order2 da COCELPA)
    //──────────────────────────────────────────────────────────────────────────────
    IF currentOrder.order2.sheetQuantity > 0 THEN
        // Se order1 não usa vincadores, order2 pode começar do índice 1
        IF currentOrder.order1.sheetQuantity > 0 AND currentOrder.order1.sheetType = SHEET_WITH_NO_SCORER THEN
            CASE currentOrder.order2.sheetQuantity OF
                1:
                    CASE currentOrder.order2.sheetType OF
                        SHEET_WITH_TWO_SCORER:
                            // Tenta posicionar conforme limites (Lógica MRBRASIL aplicada à order2)
                            IF NOT (scorerPositionArr[1] > machineConfig.scorerMaxPostionArr[3] OR
                                scorerPositionArr[2] > machineConfig.scorerMaxPostionArr[4] OR
                                scorerPositionArr[1] < machineConfig.scorerMinPostionArr[3] OR
                                scorerPositionArr[2] < machineConfig.scorerMinPostionArr[4]) THEN
                                currentOrder.generatedOrder.scorerPositionReferenceArr[3] := scorerPositionArr[1];
                                currentOrder.generatedOrder.scorerPositionReferenceArr[4] := scorerPositionArr[2];
                                currentOrder.generatedOrder.scorerEnabledArr[3] := TRUE;
                                currentOrder.generatedOrder.scorerEnabledArr[4] := TRUE;
                            ELSIF NOT (scorerPositionArr[1] > machineConfig.scorerMaxPostionArr[5] OR
                                scorerPositionArr[2] > machineConfig.scorerMaxPostionArr[6] OR
                                scorerPositionArr[1] < machineConfig.scorerMinPostionArr[5] OR
                                scorerPositionArr[2] < machineConfig.scorerMinPostionArr[6]) THEN
                                currentOrder.generatedOrder.scorerPositionReferenceArr[5] := scorerPositionArr[1];
                                currentOrder.generatedOrder.scorerPositionReferenceArr[6] := scorerPositionArr[2];
                                currentOrder.generatedOrder.scorerEnabledArr[5] := TRUE;
                                currentOrder.generatedOrder.scorerEnabledArr[6] := TRUE;
                            END_IF;
                        SHEET_WITH_FOUR_SCORER:
                            FOR i := 1 TO 4 DO
                                currentOrder.generatedOrder.scorerPositionReferenceArr[i] := scorerPositionArr[i];
                                currentOrder.generatedOrder.scorerEnabledArr[i] := TRUE;
                            END_FOR;
                    END_CASE;

                2:
                    FOR i := 1 TO 4 DO
                        currentOrder.generatedOrder.scorerPositionReferenceArr[i + 4] := scorerPositionArr[i];
                        currentOrder.generatedOrder.scorerEnabledArr[i + 4] := TRUE;
                    END_FOR;

                3:
                    FOR i := 1 TO 6 DO
                        currentOrder.generatedOrder.scorerPositionReferenceArr[i] := scorerPositionArr[i];
                        currentOrder.generatedOrder.scorerEnabledArr[i] := TRUE;
                    END_FOR;

                4, 5:
                    FOR i := 1 TO 8 DO
                        currentOrder.generatedOrder.scorerPositionReferenceArr[i] := scorerPositionArr[i];
                        currentOrder.generatedOrder.scorerEnabledArr[i] := TRUE;
                    END_FOR;
            END_CASE;

        ELSE
            // Se order1 já está ocupando ferramentas, order2 começa do índice 5
            CASE currentOrder.order2.sheetQuantity OF
                1:
                    CASE currentOrder.order2.sheetType OF
                        SHEET_WITH_TWO_SCORER:
                            currentOrder.generatedOrder.scorerPositionReferenceArr[5] := scorerPositionArr[numberOfScorersTopOrder + 1];
                            currentOrder.generatedOrder.scorerPositionReferenceArr[6] := scorerPositionArr[numberOfScorersTopOrder + 2];
                            currentOrder.generatedOrder.scorerEnabledArr[5] := TRUE;
                            currentOrder.generatedOrder.scorerEnabledArr[6] := TRUE;
                        SHEET_WITH_FOUR_SCORER:
                            FOR i := 5 TO 8 DO
                                currentOrder.generatedOrder.scorerPositionReferenceArr[i] := scorerPositionArr[i - 4];
                                currentOrder.generatedOrder.scorerEnabledArr[i] := TRUE;
                            END_FOR;
                    END_CASE;

                2:
                    FOR i := 5 TO 8 DO
                        currentOrder.generatedOrder.scorerPositionReferenceArr[i] := scorerPositionArr[i - 4];
                        currentOrder.generatedOrder.scorerEnabledArr[i] := TRUE;
                    END_FOR;

                3:
                    FOR i := 5 TO 8 DO
                        currentOrder.generatedOrder.scorerPositionReferenceArr[i] := scorerPositionArr[i - 2];
                        currentOrder.generatedOrder.scorerEnabledArr[i] := TRUE;
                    END_FOR;

                4, 5:
                    FOR i := 5 TO 8 DO
                        currentOrder.generatedOrder.scorerPositionReferenceArr[i] := scorerPositionArr[i];
                        currentOrder.generatedOrder.scorerEnabledArr[i] := TRUE;
                    END_FOR;
            END_CASE;
        END_IF;
    END_IF;
END_IF;

// Validação final (Limits check)
_checkOrderLimits();
END_ACTION

ACTION ACT_ScorerPositionSelection:

(*==============================================================================================================================
CPNTeck - Automação industrial
(c)Copyright 2022 All Rights Reserved
_______________________________________________________________________________________________________________________________
Library: N/A 
Tested with: CX5140
Engineering: Twincat 3
Restrictions: -
Requirements: N/A
Functionality: This function block offers basic functionalities for distribute the positions generated from the program to the scoring toll
Support: fabio@cpnteck.com.br
Note: Parameter comments are only available in language 'English (United States)'
_______________________________________________________________________________________________________________________________
Change log table:

Version  		| Date        			| Expert in charge  	| Changes applied
01.00.01		| 29.03.2023  		| Fabio Campion            | First released version



===============================================================================================================================*)

(*Reset the scorer enabled array*)
FOR scorerEnabledIndex := 1 TO 20 BY 1 DO

	currentOrder.generatedOrder.scorerEnabledArr[scorerEnabledIndex] := FALSE;
	scorerPositionArr[scorerEnabledIndex] := 0;
	currentOrder.generatedOrder.scorerPositionReferenceArr[scorerEnabledIndex] := 0;

END_FOR;


scorerDistributionIndex := 1;
toolDistributionIndex := 2;
scorerExecTimes := 0;

(*Calculate the number of scorers to be used in the production*)

ACT_CalculateNumberOfScorers();


(*Distribute the scorer positions*)
IF currentOrder.generatedOrder.numberOfScorers > 0 THEN

	(*Distribute the scorer position for sheets with no scorer (Only count the sheets)*)
	IF currentOrder.order1.sheetType = SHEET_WITH_NO_SCORER THEN

		FOR scorerPositionTopIndex := 1 TO currentOrder.order1.sheetQuantity BY 1 DO

			toolDistributionIndex := toolDistributionIndex + 1;

		END_FOR

	END_IF

	(*Distribute the scorer position for sheets with two scorer*)
	IF currentOrder.order1.sheetType = SHEET_WITH_TWO_SCORER THEN

		scorerExecTimes := 0;

		FOR scorerPositionTopIndex := 1 TO currentOrder.order1.sheetQuantity BY 1 DO

			scorerExecTimes := scorerExecTimes + 1;

			scorerPositionArr[scorerDistributionIndex] := toolPositionArr[toolDistributionIndex];
			scorerDistributionIndex := scorerDistributionIndex + 1;
			toolDistributionIndex := toolDistributionIndex + 1;

			scorerPositionArr[scorerDistributionIndex] := toolPositionArr[toolDistributionIndex];
			scorerDistributionIndex := scorerDistributionIndex + 1;
			toolDistributionIndex := toolDistributionIndex + 2;

		END_FOR

	END_IF

	(*Distribute the scorer position for sheets with four scorer*)
	IF currentOrder.order1.sheetType = SHEET_WITH_FOUR_SCORER THEN

		scorerExecTimes :=0;

		FOR scorerPositionTopIndex := 1 TO currentOrder.order1.sheetQuantity BY 1 DO


			scorerPositionArr[scorerDistributionIndex] := toolPositionArr[toolDistributionIndex];
			scorerDistributionIndex := scorerDistributionIndex + 1;
			toolDistributionIndex := toolDistributionIndex + 1;

			scorerPositionArr[scorerDistributionIndex] := toolPositionArr[toolDistributionIndex];
			scorerDistributionIndex := scorerDistributionIndex + 1;
			toolDistributionIndex := toolDistributionIndex + 1;

			scorerPositionArr[scorerDistributionIndex] := toolPositionArr[toolDistributionIndex];
			scorerDistributionIndex := scorerDistributionIndex + 1;
			toolDistributionIndex := toolDistributionIndex + 1;

			scorerPositionArr[scorerDistributionIndex] := toolPositionArr[toolDistributionIndex];
			scorerDistributionIndex := scorerDistributionIndex + 1;
			toolDistributionIndex := toolDistributionIndex + 2;
			

		END_FOR

	END_IF

	(*Distribute the scorer position for sheets with two scorer - bottom orderr*)
	IF currentOrder.order2.sheetType = SHEET_WITH_TWO_SCORER THEN

		scorerExecTimes := 0;

		FOR scorerPositionBottomIndex := 1 TO currentOrder.order2.sheetQuantity BY 1 DO

			scorerExecTimes := scorerExecTimes + 1;

			scorerPositionArr[scorerDistributionIndex] := toolPositionArr[toolDistributionIndex];
			scorerDistributionIndex := scorerDistributionIndex + 1;
			toolDistributionIndex := toolDistributionIndex + 1;

			scorerPositionArr[scorerDistributionIndex] := toolPositionArr[toolDistributionIndex];
			scorerDistributionIndex := scorerDistributionIndex + 1;
			toolDistributionIndex := toolDistributionIndex + 2;

		END_FOR

	END_IF

	(*Distribute the scorer position for sheets with four scorer - bottom orderr*)
	IF currentOrder.order2.sheetType = SHEET_WITH_FOUR_SCORER THEN

		scorerExecTimes := 0;

		FOR scorerPositionBottomIndex := 1 TO currentOrder.order2.sheetQuantity BY 1 DO

			scorerPositionArr[scorerDistributionIndex] := toolPositionArr[toolDistributionIndex];
			scorerDistributionIndex := scorerDistributionIndex + 1;
			toolDistributionIndex := toolDistributionIndex + 1;

			scorerPositionArr[scorerDistributionIndex] := toolPositionArr[toolDistributionIndex];
			scorerDistributionIndex := scorerDistributionIndex + 1;
			toolDistributionIndex := toolDistributionIndex + 1;

			scorerPositionArr[scorerDistributionIndex] := toolPositionArr[toolDistributionIndex];
			scorerDistributionIndex := scorerDistributionIndex + 1;
			toolDistributionIndex := toolDistributionIndex + 1;

			scorerPositionArr[scorerDistributionIndex] := toolPositionArr[toolDistributionIndex];
			scorerDistributionIndex := scorerDistributionIndex + 1;
			toolDistributionIndex := toolDistributionIndex + 2;

		END_FOR

	END_IF

END_IF

//ACT_ScorerPositionDistribution();
_scorerPositionDistribution_1();
END_ACTION

END_FUNCTION_BLOCK

// ---- Library/Machine/Slitter/FunctionBlocks/FB_ScorerHeight.TcPOU
FUNCTION_BLOCK FB_ScorerHeight
VAR_INPUT

	EN					: BOOL;
	autoManual			: BOOL;

	manualIncrement		: BOOL;
	manualDecrement		: BOOL;
	circuitBreaker		: BOOL;
	limitMax			: BOOL;
	limitMin			: BOOL;
	scorerHeightPositionSensor	: WORD;
	fluteType			: STRING;
	scorerHeightArr		: ARRAY [1..5] OF REAL;	(*Scorer height setpoint*)


END_VAR
VAR_OUTPUT

	ENO						: BOOL;
	error					: BOOL;
	positionIncrement		: BOOL;
	positionDecrement		: BOOL;
	scorerHeightMM			: REAL;				(*Scorer height position actual value in milimiters*)
	scorerHeightDifMM		: REAL;	(*Diference btween setpoint and actual value*)

END_VAR
VAR
END_VAR


(*==============================================================================================================================
CPNTeck - Automação industrial
(c)Copyright 2023 All Rights Reserved
_______________________________________________________________________________________________________________________________
Library: N/A 
Tested with: CX5140
Engineering: Twincat 2
Restrictions: -
Requirements: N/A
Functionality: This function is used control the scorer height positioning
Support: fabio@cpnteck.com.br
Note: Parameter comments are only available in language 'English (United States)'
_______________________________________________________________________________________________________________________________
Change log table:

Version  		| Date        			| Expert in charge  	| Changes applied
01.00.01		| 29.03.2023  		| Fabio Campion            | First released version



===============================================================================================================================*)

ACT_IncrementDecrement();
ACT_ScorerHeightSensor();

ACTION ACT_IncrementDecrement:
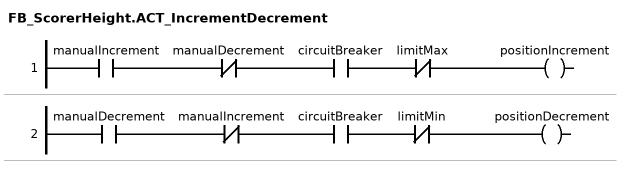
// NETWORK 1
positionIncrement := manualIncrement AND NOT manualDecrement AND circuitBreaker AND NOT limitMax;

// NETWORK 2
positionDecrement := manualDecrement AND NOT manualIncrement AND circuitBreaker AND NOT limitMin;
END_ACTION

ACTION ACT_ScorerHeightSensor:


scorerHeightMM := SCALE_R(
	X:= scorerHeightPositionSensor, 
	I_LO:= 7120, 
	I_HI:= 23880, 
	O_LO:= 3, 
	O_HI:= 0);
END_ACTION

END_FUNCTION_BLOCK

// ---- Library/Machine/Slitter/FunctionBlocks/FB_PaperDirectionControl.TcPOU
FUNCTION_BLOCK FB_PaperDirectionControl
VAR_INPUT
	
	executeCmd	: BOOL;
	allUPCmd : BOOL;
	allDownCmd : BOOL;
	invertDirection	: BOOL;
	numberOfFlaps				: INT := 27;
	flapsManualCmdArr			: ARRAY [1..27] OF hmiCommandsFlaps_TypeStruct;	
	currentOrder				: Order_TypeStruct;
	machineConfig				: slitterConfig_TypeStruct; // Slitter configuration parameters / Parâmetros do slitter

END_VAR
VAR_OUTPUT
	
	flapSolenoidArr			: ARRAY [1..27] OF BOOL;	

END_VAR


VAR
	invertDirectionOld	: BOOL;
	executeCmdOld: BOOL;
	i: INT;
END_VAR

// Trigger logic on rising edge of execute command
IF executeCmd AND NOT executeCmdOld THEN

    FOR i := 1 TO numberOfFlaps DO
        
        // 1. Level 1 Only (Upper)
        IF currentOrder.levelSelector = E_LevelSelector.eUpperOnly THEN
            flapSolenoidArr[i] := TRUE;

        // 2. Level 2 Only (Lower)
        ELSIF currentOrder.levelSelector = E_LevelSelector.eLowerOnly THEN
            flapSolenoidArr[i] := FALSE;

        // 3. Both Levels (Decision based on Order 1 Width vs Flap physical position)
        ELSIF currentOrder.levelSelector = E_LevelSelector.eBoth THEN
            
            // If flap is within the width of Order 1, it follows Order 1 direction
            IF machineConfig.arrFlapPosition[i] <= (currentOrder.generatedOrder.order1Width + currentOrder.generatedOrder.firstKnifePosition) THEN
                flapSolenoidArr[i] :=  FALSE;
            ELSE
                // Otherwise it follows Order 2 direction
                flapSolenoidArr[i] :=  TRUE;
            END_IF;

        END_IF;
    END_FOR;

END_IF;
// Update edge detection memory
executeCmdOld := executeCmd;

// Global Overrides (Master Up / Master Down)
// These run regardless of the executeCmd rising edge if triggered
IF allUPCmd THEN
    FOR i := 1 TO 27 DO flapSolenoidArr[i] := TRUE; END_FOR;
ELSIF allDownCmd THEN
    FOR i := 1 TO 27 DO flapSolenoidArr[i] := FALSE; END_FOR;
	
END_IF;

// Manual HMI Control Override (If enabled in the HMI command structure)
FOR i := 1 TO 27 DO
    IF flapsManualCmdArr[i].upCmd THEN
        flapSolenoidArr[i] := TRUE;
    END_IF;
	
    IF flapsManualCmdArr[i].downCmd THEN
        flapSolenoidArr[i] := FALSE;
    END_IF;	
	
END_FOR;

//Invert flap direction
IF invertDirection AND NOT invertDirectionOld THEN
	
	// Loop through all flaps and flip their current solenoid state
	FOR i := 1 TO numberOfFlaps DO
		flapSolenoidArr[i] := NOT flapSolenoidArr[i];
	END_FOR;

END_IF
invertDirectionOld := invertDirection;

END_FUNCTION_BLOCK

// ---- Library/Machine/Rotary knife/Function Block/FB_RotaryKnife.TcPOU
FUNCTION_BLOCK FB_RotaryKnife

VAR_INPUT
    //────────────────────────────────────────────
    // SAFETY / GUARDS / INTERLOCKS
    //────────────────────────────────────────────
    resetCmd                        : BOOL;
    safetyFeedback                  : BOOL;

    exitGuardClosed                   : BOOL;
    infeedGuardClosed                 : BOOL;
    exhaustPressurized              : BOOL;
    exhaustDepressurized            : BOOL;

    //────────────────────────────────────────────
    // UPPER KNIFE — COMMANDS / SENSORS / STATUS
    //────────────────────────────────────────────
    upperKnifePowerONCmd            : BOOL;
    upperKnifePowerOFFCmd           : BOOL;

    upperKnifeJogFwCmd              : BOOL;
    upperKnifeJogRevCmd             : BOOL;
    upperKnifeCutCmd                : BOOL;

    upperKnifeHomeSensor            : BOOL;
    upperKnifePaperSensor           : BOOL;

    upperKnifeGuardClosed           : BOOL;
    upperKnifeOilLevelLow           : BOOL;
    upperKnifeJamDetected           : BOOL;

    upperKnifeInfeedDrvOK           : BOOL;
    upperKnifeOutfeedDrvOK          : BOOL;
    upperKnifeMainDrvOK             : BOOL;
    upperKnifeSlave1DrvOK           : BOOL;
    upperKnifeSlave2DrvOK           : BOOL;
	upperKnifeResetTotalOfCuts		: BOOL;
	
    //────────────────────────────────────────────
    // LOWER KNIFE — COMMANDS / SENSORS / STATUS
    //────────────────────────────────────────────
    lowerKnifePowerONCmd            : BOOL;
    lowerKnifePowerOFFCmd           : BOOL;

    lowerKnifeJogFwCmd              : BOOL;
    lowerKnifeJogRevCmd             : BOOL;
    lowerKnifeCutCmd                : BOOL;

    lowerKnifeHomeSensor            : BOOL;
    lowerKnifePaperSensor           : BOOL;

    lowerKnifeGuardClosed           : BOOL;
    lowerKnifeOilLevelLow           : BOOL;
    lowerKnifeJamDetected           : BOOL;

    lowerKnifeInfeedDrvOK           : BOOL;
    lowerKnifeOutfeedDrvOK          : BOOL;
    lowerKnifeMainDrvOK             : BOOL;
    lowerKnifeSlave1DrvOK           : BOOL;
    lowerKnifeSlave2DrvOK           : BOOL;
	lowerKnifeResetTotalOfCuts		: BOOL;

    //────────────────────────────────────────────
    // COMMON / LINE / ENCODER / CONFIG
    //────────────────────────────────────────────
    lineSpeedMPM                    : REAL;
    aocSpeedMPM                     : REAL;
    aocRunning                      : BOOL;

    measuringWheelPaperPresence     : BOOL;

    encoderSwitchAutoMan            : BOOL := TRUE;


    machineConfigLowerKnife : rotaryKnifeConfig_TypeStruct;
    machineConfigUpperKnife : rotaryKnifeConfig_TypeStruct;
	
    currentOrder              : Order_TypeStruct; // Active order / Ordem atual
		
END_VAR
VAR_OUTPUT
    //────────────────────────────────────────────
    // GENERAL / ALARMS
    //────────────────────────────────────────────
    alarmActive                     : BOOL;

    //────────────────────────────────────────────
    // DISPLAY LINE SPEED
    //────────────────────────────────────────────
    lineSpeed                     : REAL;
    lineSpeedStacker                     : REAL;
	
	
	
    //────────────────────────────────────────────
    // External control
    //────────────────────────────────────────────	
	lineStop						: BOOL;
	lineSpeedInc					: BOOL;
	lineSpeedDec					: BOOL;
	startOutfeedConveyor			: BOOL;
	
	
    //────────────────────────────────────────────
    // UPPER KNIFE — ENABLE / RUN
    //────────────────────────────────────────────
    upperKnifeEnable                : BOOL;
    upperKnifeInFeedRun             : BOOL;
    upperKnifeOutFeedRun            : BOOL;
    upperKnifeSlave1Run             : BOOL;
    upperKnifeSlave2Run             : BOOL;

    //────────────────────────────────────────────
    // UPPER KNIFE — MOTION
    //────────────────────────────────────────────
    upperKnifeJogFw                 : BOOL;
    upperKnifeJogRev                : BOOL;
    upperKnifeCut                   : BOOL;
    upperKnifeHome                  : BOOL;
    upperKnifeHomeSensorPulse       : BOOL;
	upperEnbVirtualMaster			: BOOL;
	
    upperKnifeReset                 : BOOL;

    upperKnifeInFeedDriveRef        : REAL;
    upperKnifeOutFeedDriveRef       : REAL;

    upperKnifeEncoderSwitch         : BOOL;
    upperKnifeLubrification         : BOOL;
	
	
	
	upperKnifeSpeedLimit			 : BOOL;
	upperKnifeSpeedCurveActive		 : INT;
	upperKnifeMaximumSpeedActive 	 : REAL;
    //────────────────────────────────────────────
    // LOWER KNIFE — ENABLE / RUN
    //────────────────────────────────────────────
    lowerKnifeEnable                : BOOL;
    lowerKnifeInFeedRun             : BOOL;
    lowerKnifeOutFeedRun            : BOOL;
    lowerKnifeSlave1Run             : BOOL;
    lowerKnifeSlave2Run             : BOOL;

    //────────────────────────────────────────────
    // LOWER KNIFE — MOTION
    //────────────────────────────────────────────
    lowerKnifeJogFw                 : BOOL;
    lowerKnifeJogRev                : BOOL;
    lowerKnifeCut                   : BOOL;
    lowerKnifeHome                  : BOOL;
    lowerKnifeHomeSensorPulse       : BOOL;
	lowerEnbVirtualMaster			: BOOL;

    lowerKnifeReset                 : BOOL;

    lowerKnifeInFeedDriveRef        : REAL;
    lowerKnifeOutFeedDriveRef       : REAL;

    lowerKnifeEncoderSwitch         : BOOL;
    lowerKnifeLubrification         : BOOL;

	
	lowerKnifeSpeedLimit			 : BOOL;
	lowerKnifeSpeedCurveActive		 : INT;
	lowerKnifeMaximumSpeedActive 	 : REAL;


	measuringWheelSolenoid			: BOOL;
	
    //────────────────────────────────────────────
    // HMI STATUS
    //────────────────────────────────────────────
    upperKnifeHmiStatus                       : rotaryKnifeHmiStatus_TypeStruct;
    lowerKnifeHmiStatus                       : rotaryKnifeHmiStatus_TypeStruct;
	
END_VAR
VAR
	
    instFB_Gen_SRamp           : FB_Gen_SRamp;

    //────────────────────────────────────────────
    // UPPER KNIFE — INTERNAL
    //────────────────────────────────────────────
    upperKnifeStep                  : INT := 0;
    upperKnifeAllDrivesOK           : BOOL := FALSE;
	upperKnifeReduceLineSpeed 		: BOOL;
	upperKnifeAllInterlocksOK		: BOOL;
	
	
	
    upperKnifeRtEnable              : R_TRIG;
    upperKnifeRtPowerOff            : R_TRIG;

    upperKnifeTimerReset            : TON;
    upperKnifeTimerPulse            : TON;
    upperKnifeTimerWait             : TON;
    upperKnifeTimerClear            : TON;
	instFB_SpeedLimitUpperKnife				: FB_SpeedLimit;
	instTONUpperKnifeSwichEncoderDelay	: TON;

    //────────────────────────────────────────────
    // LOWER KNIFE — INTERNAL
    //────────────────────────────────────────────
    lowerKnifeStep                  : INT := 0;
    lowerKnifeAllDrivesOK           : BOOL := FALSE;
	lowerKnifeReduceLineSpeed 		: BOOL;
	lowerKnifeAllInterlocksOK		: BOOL;
	

    lowerKnifeRtEnable              : R_TRIG;
    lowerKnifeRtPowerOff            : R_TRIG;

    lowerKnifeTimerReset            : TON;
    lowerKnifeTimerPulse            : TON;
    lowerKnifeTimerWait             : TON;
    lowerKnifeTimerClear            : TON;
	instFB_SpeedLimitLowerKnife				: FB_SpeedLimit;
	instTONLowerKnifeSwitchEncoderDelay	: TON;

    //────────────────────────────────────────────
    // MODBUS TCP
    //────────────────────────────────────────────
    instFB_MBReadRegs               : FB_MBReadRegs;
	
    instFB_MBWriteRegs              : FB_MBWriteRegs;
    instFB_MBWriteRegs1              : FB_MBWriteRegs;
	
    modbusTCPStep                   : INT;

    upperKnifeStatusWord1           : INT;
    upperKnifeStatusWord2           : INT;
    upperKnifeModbusDword           : DWORD;
    upperKnifeWriteMenu2029         : DWORD;
    upperKnifeWriteMenu2023         : DWORD;
	
    upperKnifeLineSpeed             : INT;
    upperKnifeStatusW1              : rotaryKnifeStatusWord1_TypeStruct;
    upperKnifeStatusW2              : rotaryKnifeStatusWord2_TypeStruct;

    lowerKnifeStatusWord1           : INT;
    lowerKnifeStatusWord2           : INT;
    lowerKnifeModbusDword           : DWORD;
    lowerKnifeWriteMenu2029         : DWORD;
    lowerKnifeWriteMenu2023         : DWORD;
	
    lowerKnifeLineSpeed             : INT;
    lowerKnifeStatusW1              : rotaryKnifeStatusWord1_TypeStruct;
    lowerKnifeStatusW2              : rotaryKnifeStatusWord2_TypeStruct;
	
	upperKnifeHomeSensorOld: BOOL;
	lowerKnifeHomeSensorOld: BOOL;
	
	
	virtualMasterSpeed	: INT;
	writeVirtualMasterSpeed : BOOL;
	
	
	lineSpeedMPMRamp: REAL;
	enableVirtualMaster: BOOL;
	instTOF_UpperKnifePaperSensor: TOF;
	instTOF_LowerKnifePaperSensor: TOF;
	faultDetected: BOOL;
    instTP_LineStop  : TP;
    instRtrigFault   : R_TRIG;
	
	instTONMeasuringWheelDelay: TON;
	upperLevelInfeedSpeedLimit: REAL;
	lowerLevelInfeedSpeedLimit: REAL;
	
        upperKnifeWriteMenu2023_Raw : DWORD;
        lowerKnifeWriteMenu2023_Raw : DWORD;
		
        upperKnifeReadMenu1934_Value : BOOL;
        lowerKnifeReadMenu1934_Value : BOOL;

        upperKnifeWriteMenu1934_WriteValue : WORD;
        lowerKnifeWriteMenu1934_WriteValue : WORD;
//==========================================================
    // PRE-PROCESSING TEMPORARIES (Intermediate Calculations)
    //==========================================================
    uLengthTemp             : REAL;          // Calculated Upper Sheet Length (mm)
    lLengthTemp             : REAL;          // Calculated Lower Sheet Length (mm)
    uDiamTemp               : REAL;          // Effective Upper Knife Diameter (mm)
    lDiamTemp               : REAL;          // Effective Lower Knife Diameter (mm)		
	
END_VAR

VAR PERSISTENT
	
	upperKnifeTotalOfCutsAccumulator : DINT;
    lowerKnifeTotalOfCutsAccumulator : DINT;
	
END_VAR

_00_ModbusTCP();
_01_UpperLevelControl();
_02_LowerLevelControl();
_03_LineSpeedLimit();
_04_AuxControls();
_05_DisplayVariables();
_06_TotalOfCuts();
_07_LineSpeedRamp();
_08_StopTheLineCommand();
_09_MeasuringWheel();

METHOD _00_ModbusTCP

VAR CONSTANT
    MB_TCP_PORT         : UINT := 2010;
    MB_UNIT_ID          : USINT := 11;

    MB_TMO_READ         : TIME := T#500ms;
    MB_TMO_WRITE        : TIME := T#1000ms;

    IP_UPPER_KNIFE      : STRING := '192.168.30.86';
    IP_LOWER_KNIFE      : STRING := '192.168.30.87';

	// Address = (Menu * 100) + Parameter - 1
	MBADDR_LINE_SPEED          : UINT := 16#0711; // Pr 18.10 -> (18*100)+10-1 = 1809 -> 16#0711
	MBADDR_STATUS_W1           : UINT := 16#0774; // Pr 19.09 -> (19*100)+09-1 = 1908 -> 16#0774
	MBADDR_STATUS_W2           : UINT := 16#0775; // Pr 19.10 -> (19*100)+10-1 = 1909 -> 16#0775
	MBADDR_SHEET_LEN_20_29     : UINT := 16#47EC; // Pr 20.29 -> (20*100)+29-1 = 2028 -> 16#07EC (Start)
	MBADDR_KNIFE_DIAM_20_23    : UINT := 16#47E6; // Pr 20.23 -> (20*100)+23-1 = 2022 -> 16#07E6 (32-bit)	
	
	// New Parameter Updates
	MBADDR_V_MST_SPEED_18_26   : UINT := 16#0721; // Pr 18.26 -> (18*100)+26-1 = 1825 -> 16#0721
	MBADDR_V_MST_ENB_18_45     : UINT := 16#0734; // Pr 18.45 -> (18*100)+45-1 = 1844 -> 16#0734


	//	virtualMasterSpeed	: INT;
	// writeVirtualMasterSpeed : BOOL;

	
END_VAR
CASE currentOrder.levelSelector OF

    //----------------------------------------------------------
    // SINGLE PRODUCTION: UPPER KNIFE ACTIVE
    //----------------------------------------------------------
    E_LevelSelector.eUpperOnly:
        IF currentOrder.order1.sheetLength >= 400 THEN

            // Length Calculation - Upper knife selected length
            upperKnifeHmiStatus.sheetLength := currentOrder.order1.sheetLength + machineConfig.upperKnife.lengthAdjustment;
            lowerKnifeHmiStatus.sheetLength := upperKnifeHmiStatus.sheetLength;

            upperKnifeModbusDword := REAL_TO_DWORD(upperKnifeHmiStatus.sheetLength) * 1000;
            lowerKnifeModbusDword := upperKnifeModbusDword;

            // Diameter Logic
            IF currentOrder.order1.sheetLength < (machineConfig.upperKnife.knifeDiameter * 3.141592) THEN
                uDiamTemp := (currentOrder.order1.sheetLength / 3.141592) * machineConfig.upperKnife.knifeDiameterFactor;
            ELSE
                uDiamTemp := machineConfig.upperKnife.knifeDiameter;
            END_IF;

            upperKnifeWriteMenu2023_Raw := REAL_TO_DWORD(uDiamTemp * 1000.0);
            lowerKnifeWriteMenu2023_Raw := upperKnifeWriteMenu2023_Raw;

        END_IF;


    //----------------------------------------------------------
    // SINGLE PRODUCTION: LOWER KNIFE ACTIVE
    //----------------------------------------------------------
    E_LevelSelector.eLowerOnly:
        IF currentOrder.order1.sheetLength >= 400 THEN

            // Length Calculation - Lower knife selected length
            lowerKnifeHmiStatus.sheetLength := currentOrder.order1.sheetLength + machineConfig.lowerKnife.lengthAdjustment;
            upperKnifeHmiStatus.sheetLength := lowerKnifeHmiStatus.sheetLength;

            upperKnifeModbusDword := REAL_TO_DWORD(lowerKnifeHmiStatus.sheetLength) * 1000;
            lowerKnifeModbusDword := upperKnifeModbusDword;

            // Diameter Logic
            IF currentOrder.order1.sheetLength < (machineConfig.lowerKnife.knifeDiameter * 3.141592) THEN
                uDiamTemp := (currentOrder.order1.sheetLength / 3.141592) * machineConfig.lowerKnife.knifeDiameterFactor;
            ELSE
                uDiamTemp := machineConfig.lowerKnife.knifeDiameter;
            END_IF;

            upperKnifeWriteMenu2023_Raw := REAL_TO_DWORD(uDiamTemp * 1000.0);
            lowerKnifeWriteMenu2023_Raw := upperKnifeWriteMenu2023_Raw;

        END_IF;


    //----------------------------------------------------------
    // DUAL PRODUCTION: SPLIT ORDERS
    //----------------------------------------------------------
    E_LevelSelector.eBoth:

        // Upper write only if valid
        IF currentOrder.order1.sheetLength >= 400 THEN

            // Length Calculation - Upper knife uses order1
            upperKnifeHmiStatus.sheetLength := currentOrder.order1.sheetLength + machineConfig.upperKnife.lengthAdjustment;

            upperKnifeModbusDword := REAL_TO_DWORD(upperKnifeHmiStatus.sheetLength) * 1000;

            IF currentOrder.order1.sheetLength < (machineConfig.upperKnife.knifeDiameter * 3.141592) THEN
                uDiamTemp := (currentOrder.order1.sheetLength / 3.141592) * machineConfig.upperKnife.knifeDiameterFactor;
            ELSE
                uDiamTemp := machineConfig.upperKnife.knifeDiameter;
            END_IF;

            upperKnifeWriteMenu2023_Raw := REAL_TO_DWORD(uDiamTemp * 1000.0);

        END_IF;


        // Lower write only if valid
        IF currentOrder.order2.sheetLength >= 400 THEN

            // Length Calculation - Lower knife uses order2
            lowerKnifeHmiStatus.sheetLength := currentOrder.order2.sheetLength + machineConfig.lowerKnife.lengthAdjustment;

            lowerKnifeModbusDword := REAL_TO_DWORD(lowerKnifeHmiStatus.sheetLength) * 1000;

            IF currentOrder.order2.sheetLength < (machineConfig.lowerKnife.knifeDiameter * 3.141592) THEN
                lDiamTemp := (currentOrder.order2.sheetLength / 3.141592) * machineConfig.lowerKnife.knifeDiameterFactor;
            ELSE
                lDiamTemp := machineConfig.lowerKnife.knifeDiameter;
            END_IF;

            lowerKnifeWriteMenu2023_Raw := REAL_TO_DWORD(lDiamTemp * 1000.0);

        END_IF;

END_CASE;



//==============================================================
// MODBUS TCP MASTER STATE MACHINE
//==============================================================

CASE modbusTCPStep OF
	
	// 10: UPPER - Write Knife Diameter
    00:
        upperKnifeWriteMenu2023 := SHR(upperKnifeWriteMenu2023_Raw, 16) OR SHL(upperKnifeWriteMenu2023_Raw, 16);
        instFB_MBWriteRegs(sIPAddr:= IP_UPPER_KNIFE, nTCPPort:= MB_TCP_PORT, nUnitID:= MB_UNIT_ID, nQuantity:= 2, nMBAddr:= MBADDR_KNIFE_DIAM_20_23, cbLength:= SIZEOF(upperKnifeWriteMenu2023), pSrcAddr:= ADR(upperKnifeWriteMenu2023), bExecute:= TRUE, tTimeout:= MB_TMO_WRITE);
        IF NOT instFB_MBWriteRegs.bBusy THEN instFB_MBWriteRegs(bExecute := FALSE); modbusTCPStep := 1; END_IF

    // 11: LOWER - Write Knife Diameter
    01:
        lowerKnifeWriteMenu2023 := SHR(lowerKnifeWriteMenu2023_Raw, 16) OR SHL(lowerKnifeWriteMenu2023_Raw, 16);
        instFB_MBWriteRegs(sIPAddr:= IP_LOWER_KNIFE, nTCPPort:= MB_TCP_PORT, nUnitID:= MB_UNIT_ID, nQuantity:= 2, nMBAddr:= MBADDR_KNIFE_DIAM_20_23, cbLength:= SIZEOF(lowerKnifeWriteMenu2023), pSrcAddr:= ADR(lowerKnifeWriteMenu2023), bExecute:= TRUE, tTimeout:= MB_TMO_WRITE);
        IF NOT instFB_MBWriteRegs.bBusy THEN instFB_MBWriteRegs(bExecute := FALSE); modbusTCPStep := 2; END_IF	

    // 00-05: READS (Keeping your existing logic)
    02: // UPPER - Read Line Speed
        instFB_MBReadRegs(sIPAddr:= IP_UPPER_KNIFE, nTCPPort:= MB_TCP_PORT, nUnitID:= MB_UNIT_ID, nQuantity:= 1, nMBAddr:= MBADDR_LINE_SPEED, cbLength:= SIZEOF(upperKnifeLineSpeed), pDestAddr:= ADR(upperKnifeLineSpeed), bExecute:= TRUE, tTimeout:= MB_TMO_READ);
        IF NOT instFB_MBReadRegs.bBusy THEN instFB_MBReadRegs(bExecute := FALSE); modbusTCPStep := 3; END_IF

    03: // UPPER - Read Status W1
        instFB_MBReadRegs(sIPAddr:= IP_UPPER_KNIFE, nTCPPort:= MB_TCP_PORT, nUnitID:= MB_UNIT_ID, nQuantity:= 1, nMBAddr:= MBADDR_STATUS_W1, cbLength:= SIZEOF(upperKnifeStatusWord1), pDestAddr:= ADR(upperKnifeStatusWord1), bExecute:= TRUE, tTimeout:= MB_TMO_READ);
        IF NOT instFB_MBReadRegs.bBusy THEN instFB_MBReadRegs(bExecute := FALSE); modbusTCPStep := 4; END_IF

    04: // UPPER - Read Status W2
        instFB_MBReadRegs(sIPAddr:= IP_UPPER_KNIFE, nTCPPort:= MB_TCP_PORT, nUnitID:= MB_UNIT_ID, nQuantity:= 1, nMBAddr:= MBADDR_STATUS_W2, cbLength:= SIZEOF(upperKnifeStatusWord2), pDestAddr:= ADR(upperKnifeStatusWord2), bExecute:= TRUE, tTimeout:= MB_TMO_READ);
        IF NOT instFB_MBReadRegs.bBusy THEN instFB_MBReadRegs(bExecute := FALSE); modbusTCPStep := 5; END_IF

    05: // LOWER - Read Line Speed
        instFB_MBReadRegs(sIPAddr:= IP_LOWER_KNIFE, nTCPPort:= MB_TCP_PORT, nUnitID:= MB_UNIT_ID, nQuantity:= 1, nMBAddr:= MBADDR_LINE_SPEED, cbLength:= SIZEOF(lowerKnifeLineSpeed), pDestAddr:= ADR(lowerKnifeLineSpeed), bExecute:= TRUE, tTimeout:= MB_TMO_READ);
        IF NOT instFB_MBReadRegs.bBusy THEN instFB_MBReadRegs(bExecute := FALSE); modbusTCPStep := 6; END_IF

    06: // LOWER - Read Status W1
        instFB_MBReadRegs(sIPAddr:= IP_LOWER_KNIFE, nTCPPort:= MB_TCP_PORT, nUnitID:= MB_UNIT_ID, nQuantity:= 1, nMBAddr:= MBADDR_STATUS_W1, cbLength:= SIZEOF(lowerKnifeStatusWord1), pDestAddr:= ADR(lowerKnifeStatusWord1), bExecute:= TRUE, tTimeout:= MB_TMO_READ);
        IF NOT instFB_MBReadRegs.bBusy THEN instFB_MBReadRegs(bExecute := FALSE); modbusTCPStep := 7; END_IF

    07: // LOWER - Read Status W2
        instFB_MBReadRegs(sIPAddr:= IP_LOWER_KNIFE, nTCPPort:= MB_TCP_PORT, nUnitID:= MB_UNIT_ID, nQuantity:= 1, nMBAddr:= MBADDR_STATUS_W2, cbLength:= SIZEOF(lowerKnifeStatusWord2), pDestAddr:= ADR(lowerKnifeStatusWord2), bExecute:= TRUE, tTimeout:= MB_TMO_READ);
        IF NOT instFB_MBReadRegs.bBusy THEN instFB_MBReadRegs(bExecute := FALSE); modbusTCPStep := 8; END_IF

    // 06: UPPER - Write Cut Length
    08:
        upperKnifeWriteMenu2029 := SHR(upperKnifeModbusDword, 16) OR SHL(upperKnifeModbusDword, 16);
        instFB_MBWriteRegs(sIPAddr:= IP_UPPER_KNIFE, nTCPPort:= MB_TCP_PORT, nUnitID:= MB_UNIT_ID, nQuantity:= 2, nMBAddr:= MBADDR_SHEET_LEN_20_29, cbLength:= SIZEOF(upperKnifeWriteMenu2029), pSrcAddr:= ADR(upperKnifeWriteMenu2029), bExecute:= TRUE, tTimeout:= MB_TMO_WRITE);
        IF NOT instFB_MBWriteRegs.bBusy THEN instFB_MBWriteRegs(bExecute := FALSE); modbusTCPStep := 9; END_IF

    // 07: LOWER - Write Cut Length
    09:
        lowerKnifeWriteMenu2029 := SHR(lowerKnifeModbusDword, 16) OR SHL(lowerKnifeModbusDword, 16);
        instFB_MBWriteRegs(sIPAddr:= IP_LOWER_KNIFE, nTCPPort:= MB_TCP_PORT, nUnitID:= MB_UNIT_ID, nQuantity:= 2, nMBAddr:= MBADDR_SHEET_LEN_20_29, cbLength:= SIZEOF(lowerKnifeWriteMenu2029), pSrcAddr:= ADR(lowerKnifeWriteMenu2029), bExecute:= TRUE, tTimeout:= MB_TMO_WRITE);
        IF NOT instFB_MBWriteRegs.bBusy THEN instFB_MBWriteRegs(bExecute := FALSE); modbusTCPStep := 00; END_IF
        
    // 08: UPPER - Write Master Speed
    10:
        instFB_MBWriteRegs(sIPAddr:= IP_UPPER_KNIFE, nTCPPort:= MB_TCP_PORT, nUnitID:= MB_UNIT_ID, nQuantity:= 1, nMBAddr:= MBADDR_V_MST_SPEED_18_26, cbLength:= SIZEOF(virtualMasterSpeed), pSrcAddr:= ADR(virtualMasterSpeed), bExecute:= TRUE, tTimeout:= MB_TMO_WRITE);
        IF NOT instFB_MBWriteRegs.bBusy THEN instFB_MBWriteRegs(bExecute := FALSE); modbusTCPStep :=11; END_IF  

    // 09: LOWER - Write Master Speed
    11:
        instFB_MBWriteRegs(sIPAddr:= IP_LOWER_KNIFE, nTCPPort:= MB_TCP_PORT, nUnitID:= MB_UNIT_ID, nQuantity:= 1, nMBAddr:= MBADDR_V_MST_SPEED_18_26, cbLength:= SIZEOF(virtualMasterSpeed), pSrcAddr:= ADR(virtualMasterSpeed), bExecute:= TRUE, tTimeout:= MB_TMO_WRITE);
        IF NOT instFB_MBWriteRegs.bBusy THEN instFB_MBWriteRegs(bExecute := FALSE); modbusTCPStep := 00; END_IF      
        

END_CASE

//==============================================================
// BIT UNPACKING (Status logic remains exactly as yours)
//==============================================================
// ... [Existing Unpacking Code]

//==============================================================
// BIT UNPACKING: DRIVE STATUS TO HMI/LOGIC BOOLS
// Converts raw Modbus 16-bit registers into descriptive Booleans.
//==============================================================

// --- UPPER KNIFE STATUS WORD 1 (Operational State) ---
upperKnifeStatusW1.knifeAtHomeParkPos1              := upperKnifeStatusWord1.00;
upperKnifeStatusW1.homingInProgress                 := upperKnifeStatusWord1.01;
upperKnifeStatusW1.homingComplete                   := upperKnifeStatusWord1.02;
upperKnifeStatusW1.knifeInspectionMotionInProgress  := upperKnifeStatusWord1.03;
upperKnifeStatusW1.knifeInspectionMotionComplete    := upperKnifeStatusWord1.04;
upperKnifeStatusW1.returnHomeMotionInProgress       := upperKnifeStatusWord1.05;
upperKnifeStatusW1.returnHomeMotionComplete         := upperKnifeStatusWord1.06;
upperKnifeStatusW1.jogForwardInProgress             := upperKnifeStatusWord1.07;
upperKnifeStatusW1.jogReverseInProgress             := upperKnifeStatusWord1.08;
upperKnifeStatusW1.knifeGearingOut                  := upperKnifeStatusWord1.09;
upperKnifeStatusW1.knifeRunningEngaged              := upperKnifeStatusWord1.10; // Knife actively tracking line
upperKnifeStatusW1.knifeStoppedDisengaged           := upperKnifeStatusWord1.11;
upperKnifeStatusW1.maxLineSpeedLimitCalculated      := upperKnifeStatusWord1.12;
upperKnifeStatusW1.batchMaxLineSpeedCalcInProgress  := upperKnifeStatusWord1.13;
upperKnifeStatusW1.batchMaxLineSpeedCalculated      := upperKnifeStatusWord1.14;
upperKnifeStatusW1.watchdogClockOut                 := upperKnifeStatusWord1.15; // Heartbeat from Drive

// --- LOWER KNIFE STATUS WORD 1 (Operational State) ---
lowerKnifeStatusW1.knifeAtHomeParkPos1              := lowerKnifeStatusWord1.00;
lowerKnifeStatusW1.homingInProgress                 := lowerKnifeStatusWord1.01;
lowerKnifeStatusW1.homingComplete                   := lowerKnifeStatusWord1.02;
lowerKnifeStatusW1.knifeInspectionMotionInProgress  := lowerKnifeStatusWord1.03;
lowerKnifeStatusW1.knifeInspectionMotionComplete    := lowerKnifeStatusWord1.04;
lowerKnifeStatusW1.returnHomeMotionInProgress       := lowerKnifeStatusWord1.05;
lowerKnifeStatusW1.returnHomeMotionComplete         := lowerKnifeStatusWord1.06;
lowerKnifeStatusW1.jogForwardInProgress             := lowerKnifeStatusWord1.07;
lowerKnifeStatusW1.jogReverseInProgress             := lowerKnifeStatusWord1.08;
lowerKnifeStatusW1.knifeGearingOut                  := lowerKnifeStatusWord1.09;
lowerKnifeStatusW1.knifeRunningEngaged              := lowerKnifeStatusWord1.10;
lowerKnifeStatusW1.knifeStoppedDisengaged           := lowerKnifeStatusWord1.11;
lowerKnifeStatusW1.maxLineSpeedLimitCalculated      := lowerKnifeStatusWord1.12;
lowerKnifeStatusW1.batchMaxLineSpeedCalcInProgress  := lowerKnifeStatusWord1.13;
lowerKnifeStatusW1.batchMaxLineSpeedCalculated      := lowerKnifeStatusWord1.14;
lowerKnifeStatusW1.watchdogClockOut                 := lowerKnifeStatusWord1.15;

// --- UPPER KNIFE STATUS WORD 2 (Registration & Health) ---
upperKnifeStatusW2.batchSingleShotStopInProgress    := upperKnifeStatusWord2.00;
upperKnifeStatusW2.registrationMarkMissed           := upperKnifeStatusWord2.01;
upperKnifeStatusW2.registrationWindowOpen           := upperKnifeStatusWord2.02;
upperKnifeStatusW2.registrationMarkAccepted         := upperKnifeStatusWord2.03;
upperKnifeStatusW2.onLastBatch                      := upperKnifeStatusWord2.04;
upperKnifeStatusW2.onLastCutOfLastBatch             := upperKnifeStatusWord2.05;
upperKnifeStatusW2.pls1Output                       := upperKnifeStatusWord2.06; // Programmable Limit Switch
upperKnifeStatusW2.pls2Output                       := upperKnifeStatusWord2.07;
upperKnifeStatusW2.referenceEnabled                 := upperKnifeStatusWord2.08;
upperKnifeStatusW2.driveHealthy                     := upperKnifeStatusWord2.09; // OK to run
upperKnifeStatusW2.reserved10                       := upperKnifeStatusWord2.10;
upperKnifeStatusW2.reserved11                       := upperKnifeStatusWord2.11;
upperKnifeStatusW2.userDefinedStatusBit12           := upperKnifeStatusWord2.12;
upperKnifeStatusW2.userDefinedStatusBit13           := upperKnifeStatusWord2.13;
upperKnifeStatusW2.userDefinedStatusBit14           := upperKnifeStatusWord2.14;
upperKnifeStatusW2.userDefinedStatusBit15           := upperKnifeStatusWord2.15;

// --- LOWER KNIFE STATUS WORD 2 (Registration & Health) ---
lowerKnifeStatusW2.batchSingleShotStopInProgress    := lowerKnifeStatusWord2.00;
lowerKnifeStatusW2.registrationMarkMissed           := lowerKnifeStatusWord2.01;
lowerKnifeStatusW2.registrationWindowOpen           := lowerKnifeStatusWord2.02;
lowerKnifeStatusW2.registrationMarkAccepted         := lowerKnifeStatusWord2.03;
lowerKnifeStatusW2.onLastBatch                      := lowerKnifeStatusWord2.04;
lowerKnifeStatusW2.onLastCutOfLastBatch             := lowerKnifeStatusWord2.05;
lowerKnifeStatusW2.pls1Output                       := lowerKnifeStatusWord2.06;
lowerKnifeStatusW2.pls2Output                       := lowerKnifeStatusWord2.07;
lowerKnifeStatusW2.referenceEnabled                 := lowerKnifeStatusWord2.08;
lowerKnifeStatusW2.driveHealthy                     := lowerKnifeStatusWord2.09;
lowerKnifeStatusW2.reserved10                       := lowerKnifeStatusWord2.10;
lowerKnifeStatusW2.reserved11                       := lowerKnifeStatusWord2.11;
lowerKnifeStatusW2.userDefinedStatusBit12           := lowerKnifeStatusWord2.12;
lowerKnifeStatusW2.userDefinedStatusBit13           := lowerKnifeStatusWord2.13;
lowerKnifeStatusW2.userDefinedStatusBit14           := lowerKnifeStatusWord2.14;
lowerKnifeStatusW2.userDefinedStatusBit15           := lowerKnifeStatusWord2.15;
END_METHOD

METHOD _01_UpperLevelControl
VAR_INPUT
END_VAR
(*
    upperKnifeGuardClosed           : BOOL;
    upperKnifeOilLevelLow           : BOOL;
    upperKnifeJamDetected           : BOOL;
    exitGuardClosed                   : BOOL;
    infeedGuardClosed                 : BOOL;
*)
(*
======================================================================
UPPER KNIFE — Rotary Knife Control (Upper Knife)
======================================================================
Concept:
- Power ON command starts a simple sequence:
  0  = OFF / Idle
  10 = Enable drives + follow line speed
  20 = Send HOME command for 1s
  21 = Wait for HomingComplete status before running infeed/outfeed
  40 = Normal operation (cut enabled when command + paper present)

Rule:
- When the upper knife is powered ON, infeed/outfeed speed references
  must follow lineSpeedMPM.
======================================================================
*)

//==============================================================
// 1) RESET PULSE (2s) + EDGE DETECTION
//==============================================================
upperKnifeTimerReset(IN := resetCmd, PT := T#2S);
upperKnifeReset := upperKnifeTimerReset.Q;

upperKnifeRtEnable(CLK := upperKnifePowerONCmd);
upperKnifeRtPowerOff(CLK := upperKnifePowerOFFCmd);

//==============================================================
// 2) DRIVE / SAFETY STATUS (AGGREGATION)
//==============================================================
upperKnifeAllDrivesOK := upperKnifeInfeedDrvOK  AND
                         upperKnifeOutfeedDrvOK AND
                         upperKnifeMainDrvOK    AND
                         upperKnifeSlave1DrvOK  AND
                         upperKnifeSlave2DrvOK;

upperKnifeHomeSensorPulse := upperKnifeHomeSensor;

upperKnifeAllInterlocksOK := infeedGuardClosed AND
							 exitGuardClosed AND
							 upperKnifeGuardClosed AND
							 upperKnifeOilLevelLow AND NOT
							 upperKnifeJamDetected;
				

//==============================================================
// 3) START SEQUENCE CONDITION
//==============================================================
// Start only if:
// - Rising edge on Power ON
// - Sequence is idle
// - Safety chain OK
// - All drives OK
// - No reset pulse active
IF upperKnifeRtEnable.Q
   AND (upperKnifeStep = 0)
   AND safetyFeedback
   AND upperKnifeAllDrivesOK
   AND NOT upperKnifeReset THEN

    upperKnifeStep := 10;
END_IF

//==============================================================
// 4) SEQUENCE STATE MACHINE
//==============================================================
CASE upperKnifeStep OF

    //==========================================================
    // 0 — OFF / IDLE
    //==========================================================
    0:
        // Commands OFF
        upperKnifeEnable      := FALSE;
        upperKnifeSlave1Run   := FALSE;
        upperKnifeSlave2Run   := FALSE;
        upperKnifeInFeedRun   := FALSE;
        upperKnifeOutFeedRun  := FALSE;

        // Motion / actions OFF
        upperKnifeJogFw       := FALSE;
        upperKnifeJogRev      := FALSE;
        upperKnifeHome        := FALSE;
        upperKnifeCut         := FALSE;

        // References = 0
        upperKnifeInFeedDriveRef  := 0.0;
        upperKnifeOutFeedDriveRef := 0.0;

    //==========================================================
    // 10 — ENABLE DRIVES + FOLLOW LINE SPEED
    //==========================================================
    10:
        upperKnifeEnable      := TRUE;
        upperKnifeSlave1Run   := TRUE;
        upperKnifeSlave2Run   := TRUE;

        // Follow line speed immediately when powered ON
        upperKnifeInFeedDriveRef  := lineSpeedMPM;
        upperKnifeOutFeedDriveRef := lineSpeedMPM;

        // Next step: issue homing pulse
        upperKnifeStep := 20;

    //==========================================================
    // 20 — HOME COMMAND PULSE (1s)
    //==========================================================
    20:
        // Command home for 1 second
        upperKnifeHome := TRUE;

        upperKnifeTimerPulse(IN := TRUE, PT := T#1S);
        IF upperKnifeTimerPulse.Q THEN
            upperKnifeHome := FALSE;
            upperKnifeTimerPulse(IN := FALSE);
            upperKnifeStep := 21;
        END_IF

    //==========================================================
    // 21 — WAIT HOMING COMPLETE
    //==========================================================
    21:
        // Start infeed/outfeed only after homing is complete
//        IF upperKnifeStatusW1.homingComplete THEN
            upperKnifeInFeedRun  := TRUE;
            upperKnifeOutFeedRun := TRUE;
            upperKnifeStep := 40;
//        END_IF

    //==========================================================
    // 40 — NORMAL OPERATION
    //==========================================================
    40:
	
        upperKnifeJogFw       := upperKnifeJogFwCmd;
        upperKnifeJogRev      := upperKnifeJogRevCmd;	
	

		instTOF_UpperKnifePaperSensor(IN := upperKnifePaperSensor, PT:= T#30M);
		
	
		IF instTOF_UpperKnifePaperSensor.Q OR lineSpeedMPM > 5 THEN
		
			upperKnifeInFeedDriveRef := LIMIT(machineConfigUpperKnife.minLineSpeed,
											  lineSpeedMPMRamp,
											  upperLevelInfeedSpeedLimit) * machineConfigUpperKnife.infeedRollSpeedOffset;		
				
			upperKnifeOutFeedDriveRef := LIMIT(machineConfigUpperKnife.minLineSpeed,
											  lineSpeedMPMRamp,
											  999) * machineConfigUpperKnife.outfeedRollSpeedOffset;
		ELSE
	
			upperKnifeInFeedDriveRef := 0;				
			upperKnifeOutFeedDriveRef := 0;
		
		END_IF								  

        // Enable cut only when commanded and paper present
        upperKnifeCut := (upperKnifeCutCmd AND upperKnifePaperSensor);
		
		
		IF NOT measuringWheelPaperPresence THEN
			
			upperLevelInfeedSpeedLimit := upperKnifeMaximumSpeedActive;
			
		ELSE
		
			upperLevelInfeedSpeedLimit := 999;	
		
		END_IF		

END_CASE

//==============================================================
// 5) GLOBAL INTERLOCK — IMMEDIATE STOP
//==============================================================
// Immediate stop on any of these conditions:
// - Safety chain not OK
// - Any drive not OK
// - Power OFF command rising edge
IF (NOT safetyFeedback)
   OR (NOT upperKnifeAllDrivesOK)
   OR upperKnifeRtPowerOff.Q THEN

    upperKnifeStep := 0;

    upperKnifeEnable      := FALSE;
    upperKnifeSlave1Run   := FALSE;
    upperKnifeSlave2Run   := FALSE;
    upperKnifeInFeedRun   := FALSE;
    upperKnifeOutFeedRun  := FALSE;

    upperKnifeJogFw       := FALSE;
    upperKnifeJogRev      := FALSE;
    upperKnifeHome        := FALSE;
    upperKnifeCut         := FALSE;

    upperKnifeInFeedDriveRef  := 0.0;
    upperKnifeOutFeedDriveRef := 0.0;

    // Reset internal timers for a clean restart
    upperKnifeTimerWait(IN := FALSE);
    upperKnifeTimerPulse(IN := FALSE);
    upperKnifeTimerClear(IN := FALSE);
    upperKnifeTimerReset(IN := FALSE);
END_IF


//Start Lubrification pump
upperKnifeLubrification := upperKnifeEnable;


//==============================================================
// ENCODER SELECTION — UPPER KNIFE
//==============================================================
// Rules:
// - encoderSwitchAutoMan = FALSE → ALWAYS use machine encoder
// - encoderSwitchAutoMan = TRUE  → automatic selection based on paper presence
//==============================================================


    //----------------------------------------------------------
    // AUTO MODE
    //----------------------------------------------------------
    IF NOT measuringWheelPaperPresence THEN
        // No paper → immediate fallback to measuring wheel encoder
        upperKnifeEncoderSwitch := TRUE;

        // Reset delay timer
        instTONUpperKnifeSwichEncoderDelay.IN := FALSE;

    ELSE
        // Paper present → start delay before switching
        instTONUpperKnifeSwichEncoderDelay.IN := TRUE;

        // Switch only after delay elapsed
        IF instTONUpperKnifeSwichEncoderDelay.Q THEN
				
			upperKnifeEncoderSwitch := FALSE;

        END_IF
		
    END_IF


//--------------------------------------------------------------
// TIMER EXECUTION (ALWAYS CALLED)
//--------------------------------------------------------------
instTONUpperKnifeSwichEncoderDelay(
    PT := machineConfigUpperKnife.switchEncoderDelay
);
END_METHOD

METHOD _02_LowerLevelControl
VAR_INPUT
END_VAR
(*

    //----------------------------------------------------------
    // AUTO MODE
    //----------------------------------------------------------
    IF NOT measuringWheelPaperPresence THEN
        // No paper → immediate fallback to measuring wheel encoder
        upperKnifeEncoderSwitch := TRUE;

        // Reset delay timer
        instTONUpperKnifeSwichEncoderDelay.IN := FALSE;

    ELSE
        // Paper present → start delay before switching
        instTONUpperKnifeSwichEncoderDelay.IN := TRUE;

        // Switch only after delay elapsed
        IF instTONUpperKnifeSwichEncoderDelay.Q THEN
				
			upperKnifeEncoderSwitch := FALSE;

        END_IF
		
    END_IF

*)

(*
    //----------------------------------------------------------
    // AUTO MODE
    //----------------------------------------------------------
    IF NOT measuringWheelPaperPresence THEN
        // No paper → immediate fallback to measuring wheel encoder
        lowerEnbVirtualMaster := TRUE;

        // Reset delay timer
        instTONLowerKnifeSwitchEncoderDelay.IN := FALSE;

    ELSE
        // Paper present → start delay before switching
        instTONLowerKnifeSwitchEncoderDelay.IN := TRUE;

        // Switch only after delay elapsed
        IF instTONLowerKnifeSwitchEncoderDelay.Q THEN
            lowerEnbVirtualMaster := FALSE;
        END_IF
    END_IF


*)
(*
======================================================================
LOWER KNIFE — Rotary Knife Control (Lower Knife)
======================================================================
Concept:
- Power ON command starts a simple sequence:
  0  = OFF / Idle
  10 = Enable drives + follow line speed
  20 = Send HOME command for 1s
  21 = Wait for HomingComplete status before running infeed/outfeed
  40 = Normal operation (cut enabled when command + paper present)

Rule:
- When the lower knife is powered ON, infeed/outfeed speed references
  must follow lineSpeedMPM.
======================================================================
*)

//==============================================================
// 1) RESET PULSE (2s) + EDGE DETECTION
//==============================================================
lowerKnifeTimerReset(IN := resetCmd, PT := T#2S);
lowerKnifeReset := lowerKnifeTimerReset.Q;

lowerKnifeRtEnable(CLK := lowerKnifePowerONCmd);
lowerKnifeRtPowerOff(CLK := lowerKnifePowerOFFCmd);

//==============================================================
// 2) DRIVE / SAFETY STATUS (AGGREGATION)
//==============================================================
lowerKnifeAllDrivesOK := lowerKnifeInfeedDrvOK  AND
                         lowerKnifeOutfeedDrvOK AND
                         lowerKnifeMainDrvOK    AND
                         lowerKnifeSlave1DrvOK  AND
                         lowerKnifeSlave2DrvOK;

lowerKnifeHomeSensorPulse := lowerKnifeHomeSensor;

// NOTE: keep the same logic structure you used on upper knife.
// If your signals mean "LOW" = fault, consider inverting oil level here.
// (This is copied exactly from your upper knife reference.)
lowerKnifeAllInterlocksOK := infeedGuardClosed AND
							 exitGuardClosed AND
							 lowerKnifeGuardClosed AND
                             lowerKnifeOilLevelLow AND NOT
                             lowerKnifeJamDetected;

//==============================================================
// 3) START SEQUENCE CONDITION
//==============================================================
// Start only if:
// - Rising edge on Power ON
// - Sequence is idle
// - Safety chain OK
// - All drives OK
// - No reset pulse active
IF lowerKnifeRtEnable.Q
   AND (lowerKnifeStep = 0)
   AND safetyFeedback
   AND lowerKnifeAllDrivesOK
   AND NOT lowerKnifeReset THEN

    lowerKnifeStep := 10;
END_IF

//==============================================================
// 4) SEQUENCE STATE MACHINE
//==============================================================
CASE lowerKnifeStep OF

    //==========================================================
    // 0 — OFF / IDLE
    //==========================================================
    0:
        // Commands OFF
        lowerKnifeEnable      := FALSE;
        lowerKnifeSlave1Run   := FALSE;
        lowerKnifeSlave2Run   := FALSE;
        lowerKnifeInFeedRun   := FALSE;
        lowerKnifeOutFeedRun  := FALSE;

        // Motion / actions OFF
        lowerKnifeJogFw       := FALSE;
        lowerKnifeJogRev      := FALSE;
        lowerKnifeHome        := FALSE;
        lowerKnifeCut         := FALSE;

        // References = 0
        lowerKnifeInFeedDriveRef  := 0.0;
        lowerKnifeOutFeedDriveRef := 0.0;

    //==========================================================
    // 10 — ENABLE DRIVES + FOLLOW LINE SPEED
    //==========================================================
    10:
        lowerKnifeEnable      := TRUE;
        lowerKnifeSlave1Run   := TRUE;
        lowerKnifeSlave2Run   := TRUE;
		
        // Follow line speed immediately when powered ON
        lowerKnifeInFeedDriveRef  := lineSpeedMPM;
        lowerKnifeOutFeedDriveRef := lineSpeedMPM;

        // Next step: issue homing pulse
        lowerKnifeStep := 20;

    //==========================================================
    // 20 — HOME COMMAND PULSE (1s)
    //==========================================================
    20:
        // Command home for 1 second
        lowerKnifeHome := TRUE;

        lowerKnifeTimerPulse(IN := TRUE, PT := T#1S);
        IF lowerKnifeTimerPulse.Q THEN
            lowerKnifeHome := FALSE;
            lowerKnifeTimerPulse(IN := FALSE);
            lowerKnifeStep := 21;
        END_IF

